SPLINE
SPL {X  -165.650, Y  +465.900, Z    +0.000, E1   -37.888, E3 +418401.268}
SPL {X  -165.650, Y  +471.256, Z    +0.000, E1   -37.789, E3 +418415.836}
SPL {X  -165.650, Y  +475.981, Z    +0.000, E1   -37.909, E3 +418427.559}
SPL {X  -165.650, Y  +481.142, Z    +0.000, E1   -37.875, E3 +418441.379}
SPL {X  -165.650, Y  +485.415, Z    +0.000, E1   -37.930, E3 +418452.144}
SPL {X  -165.650, Y  +488.381, Z    +0.000, E1   -37.932, E3 +418459.911}
SPL {X  -165.650, Y  +492.473, Z    +0.000, E1   -37.882, E3 +418471.081}
SPL {X  -165.650, Y  +496.967, Z    +0.000, E1   -37.731, E3 +418483.788}
SPL {X  -165.650, Y  +502.007, Z    +0.000, E1   -37.899, E3 +418496.077}
SPL {X  -165.650, Y  +506.838, Z    +0.000, E1   -38.018, E3 +418507.973}
SPL {X  -165.650, Y  +510.962, Z    +0.000, E1   -37.876, E3 +418519.687}
SPL {X  -165.650, Y  +513.924, Z    +0.000, E1   -37.557, E3 +418529.355}
SPL {X  -165.650, Y  +519.541, Z    +0.000, E1   -37.994, E3 +418541.689}
SPL {X  -165.650, Y  +524.168, Z    +0.000, E1   -37.816, E3 +418554.745}
SPL {X  -165.650, Y  +528.532, Z    +0.000, E1   -37.895, E3 +418565.811}
SPL {X  -165.650, Y  +532.864, Z    +0.000, E1   -37.846, E3 +418577.452}
SPL {X  -165.650, Y  +537.279, Z    +0.000, E1   -37.980, E3 +418588.275}
SPL {X  -165.650, Y  +540.651, Z    +0.000, E1   -37.651, E3 +418599.077}
SPL {X  -165.650, Y  +545.726, Z    +0.000, E1   -37.963, E3 +418610.643}
SPL {X  -165.650, Y  +550.427, Z    +0.000, E1   -37.784, E3 +418624.061}
SPL {X  -165.650, Y  +554.659, Z    +0.000, E1   -37.927, E3 +418634.245}
SPL {X  -165.650, Y  +557.856, Z    +0.000, E1   -37.998, E3 +418642.195}
SPL {X  -165.650, Y  +562.748, Z    +0.000, E1   -37.890, E3 +418655.937}
SPL {X  -165.650, Y  +567.848, Z    +0.000, E1   -37.954, E3 +418668.710}
SPL {X  -165.650, Y  +571.305, Z    +0.000, E1   -37.718, E3 +418679.371}
SPL {X  -165.650, Y  +577.754, Z    +0.000, E1   -38.006, E3 +418694.662}
SPL {X  -165.650, Y  +583.042, Z    +0.000, E1   -37.879, E3 +418709.206}
SPL {X  -165.650, Y  +587.643, Z    +0.000, E1   -37.879, E3 +418721.284}
SPL {X  -165.650, Y  +592.833, Z    +0.000, E1   -37.896, E3 +418734.932}
SPL {X  -165.650, Y  +597.119, Z    +0.000, E1   -37.642, E3 +418747.661}
SPL {X  -165.650, Y  +602.808, Z    +0.000, E1   -37.983, E3 +418760.668}
SPL {X  -165.650, Y  +607.937, Z    +0.000, E1   -37.862, E3 +418774.829}
SPL {X  -165.650, Y  +614.056, Z    +0.000, E1   -37.933, E3 +418790.600}
SPL {X  -165.650, Y  +619.142, Z    +0.000, E1   -37.954, E3 +418803.618}
SPL {X  -165.650, Y  +622.884, Z    +0.000, E1   -37.770, E3 +418814.661}
SPL {X  -165.650, Y  +628.759, Z    +0.000, E1   -37.993, E3 +418828.831}
SPL {X  -165.650, Y  +633.686, Z    +0.000, E1   -37.760, E3 +418843.106}
SPL {X  -165.650, Y  +639.918, Z    +0.000, E1   -37.892, E3 +418858.915}
SPL {X  -165.650, Y  +645.851, Z    +0.000, E1   -37.854, E3 +418874.567}
SPL {X  -165.650, Y  +650.450, Z    +0.000, E1   -37.924, E3 +418886.207}
SPL {X  -165.650, Y  +654.711, Z    +0.000, E1   -37.888, E3 +418897.641}
SPL {X  -165.650, Y  +660.285, Z    +0.000, E1   -37.928, E3 +418912.159}
SPL {X  -165.650, Y  +665.663, Z    +0.000, E1   -37.913, E3 +418926.247}
SPL {X  -165.650, Y  +669.913, Z    +0.000, E1   -37.905, E3 +418937.449}
SPL {X  -165.650, Y  +674.729, Z    +0.000, E1   -37.860, E3 +418950.458}
SPL {X  -165.591, Y  +679.928, Z    +0.000, E1   -37.818, E3 +418964.375}
SPL {X  -165.340, Y  +685.624, Z    +0.000, E1   -37.900, E3 +418978.910}
SPL {X  -165.010, Y  +690.051, Z    +0.000, E1   -37.675, E3 +418991.841}
SPL {X  -164.652, Y  +693.652, Z    +0.000, E1   -37.750, E3 +419000.771}
SPL {X  -164.143, Y  +697.797, Z    +0.000, E1   -37.636, E3 +419012.591}
SPL {X  -163.447, Y  +702.423, Z    +0.000, E1   -37.496, E3 +419025.399}
SPL {X  -162.809, Y  +706.049, Z    +0.000, E1   -37.384, E3 +419035.669}
SPL {X  -161.803, Y  +710.992, Z    +0.000, E1   -37.315, E3 +419049.134}
SPL {X  -160.993, Y  +714.501, Z    +0.000, E1   -36.839, E3 +419061.011}
SPL {X  -159.156, Y  +721.427, Z    +0.000, E1   -38.526, E3 +419069.089}
SPL {X  -144.831, Y  +755.898, Z    +0.000, E1   -42.981, E3 +419130.505}
ENDSPLINE

SPLINE
SPL {X  -153.047, Y  +738.876, Z    +0.000, E1   -33.363, E3 +419212.720}
SPL {X  -162.649, Y  +706.888, Z    +0.000, E1   -19.911, E3 +419202.081}
SPL {X  -165.011, Y  +690.033, Z    +0.000, E1   -11.292, E3 +419198.316}
SPL {X  -165.581, Y  +680.273, Z    +0.000, E1    -5.775, E3 +419194.114}
SPL {X  -165.650, Y  +674.660, Z    +0.000, E1    -2.196, E3 +419194.781}
SPL {X  -165.650, Y  +669.932, Z    +0.000, E1    +1.173, E3 +419193.357}
SPL {X  -165.650, Y  +665.412, Z    +0.000, E1    +4.953, E3 +419192.537}
SPL {X  -165.650, Y  +660.335, Z    +0.000, E1    +9.682, E3 +419193.054}
SPL {X  -165.650, Y  +650.970, Z    +0.000, E1   +18.783, E3 +419193.602}
SPL {X  -165.650, Y  +637.823, Z    +0.000, E1   +39.473, E3 +419173.703}
SPL {X  -165.650, Y  +613.283, Z    +0.000, E1   +49.826, E3 +419189.271}
SPL {X  -165.650, Y  +609.693, Z    +0.000, E1   +42.113, E3 +419217.405}
SPL {X  -165.650, Y  +571.120, Z    +0.000, E1   +47.704, E3 +419262.214}
ENDSPLINE

SPLINE
SPL {X  -165.650, Y  +586.477, Z    +0.000, E1   +39.172, E3 +419278.758}
ENDSPLINE

SPLINE
SPL {X  -165.650, Y  +581.917, Z    +0.000, E1   +39.019, E3 +419291.160}
SPL {X  -165.650, Y  +577.218, Z    +0.000, E1   +38.911, E3 +419303.701}
SPL {X  -165.650, Y  +572.890, Z    +0.000, E1   +39.033, E3 +419313.838}
SPL {X  -165.650, Y  +569.005, Z    +0.000, E1   +38.999, E3 +419323.929}
SPL {X  -165.650, Y  +564.604, Z    +0.000, E1   +38.986, E3 +419335.065}
SPL {X  -165.650, Y  +560.333, Z    +0.000, E1   +38.995, E3 +419345.830}
SPL {X  -165.650, Y  +556.690, Z    +0.000, E1   +39.061, E3 +419354.549}
SPL {X  -165.650, Y  +552.186, Z    +0.000, E1   +39.063, E3 +419366.067}
SPL {X  -165.650, Y  +547.091, Z    +0.000, E1   +39.070, E3 +419378.727}
SPL {X  -165.650, Y  +526.098, Z    +0.000, E1   +45.792, E3 +419385.794}
SPL {X  -165.650, Y  +510.223, Z    +0.000, E1   +49.521, E3 +419393.191}
SPL {X  -165.650, Y  +505.315, Z    +0.000, E1   +48.718, E3 +419407.000}
SPL {X  -165.650, Y  +499.987, Z    +0.000, E1   +47.980, E3 +419420.786}
SPL {X  -165.650, Y  +497.138, Z    +0.000, E1   +47.280, E3 +419430.279}
SPL {X  -165.650, Y  +493.273, Z    +0.000, E1   +46.518, E3 +419442.260}
SPL {X  -165.650, Y  +489.140, Z    +0.000, E1   +45.675, E3 +419455.387}
SPL {X  -165.650, Y  +485.420, Z    +0.000, E1   +44.711, E3 +419468.606}
SPL {X  -165.650, Y  +480.756, Z    +0.000, E1   +43.779, E3 +419484.084}
SPL {X  -165.650, Y  +475.837, Z    +0.000, E1   +42.787, E3 +419500.545}
SPL {X  -165.650, Y  +472.413, Z    +0.000, E1   +41.852, E3 +419513.660}
SPL {X  -165.650, Y  +469.721, Z    +0.000, E1   +41.361, E3 +419522.686}
SPL {X  -165.650, Y  +467.130, Z    +0.000, E1   +40.624, E3 +419533.368}
SPL {X  -165.650, Y  +463.869, Z    +0.000, E1   +39.839, E3 +419545.836}
SPL {X  -165.650, Y  +462.171, Z    +0.000, E1   +38.860, E3 +419556.015}
SPL {X  -165.650, Y  +457.119, Z    +0.000, E1   +39.087, E3 +419567.393}
SPL {X  -165.650, Y  +452.884, Z    +0.000, E1   +39.185, E3 +419577.441}
SPL {X  -165.650, Y  +449.593, Z    +0.000, E1   +38.852, E3 +419587.736}
SPL {X  -165.650, Y  +445.147, Z    +0.000, E1   +39.088, E3 +419597.558}
SPL {X  -165.650, Y  +439.751, Z    +0.000, E1   +39.254, E3 +419610.175}
SPL {X  -165.650, Y  +435.510, Z    +0.000, E1   +39.051, E3 +419621.987}
SPL {X  -165.650, Y  +430.832, Z    +0.000, E1   +39.105, E3 +419633.443}
SPL {X  -165.650, Y  +426.072, Z    +0.000, E1   +39.194, E3 +419644.866}
SPL {X  -165.650, Y  +422.372, Z    +0.000, E1   +38.952, E3 +419655.602}
SPL {X  -165.650, Y  +417.591, Z    +0.000, E1   +39.157, E3 +419666.455}
SPL {X  -165.650, Y  +412.842, Z    +0.000, E1   +39.072, E3 +419678.954}
SPL {X  -165.650, Y  +407.612, Z    +0.000, E1   +39.068, E3 +419692.127}
SPL {X  -165.650, Y  +402.767, Z    +0.000, E1   +39.122, E3 +419703.982}
SPL {X  -165.650, Y  +398.352, Z    +0.000, E1   +39.113, E3 +419715.135}
SPL {X  -165.650, Y  +393.915, Z    +0.000, E1   +39.126, E3 +419726.212}
SPL {X  -165.650, Y  +389.523, Z    +0.000, E1   +39.115, E3 +419737.322}
SPL {X  -165.650, Y  +384.404, Z    +0.000, E1   +39.147, E3 +419750.058}
SPL {X  -165.650, Y  +380.058, Z    +0.000, E1   +39.073, E3 +419761.345}
SPL {X  -165.624, Y  +375.547, Z    +0.000, E1   +39.047, E3 +419772.944}
SPL {X  -165.438, Y  +370.129, Z    +0.000, E1   +39.090, E3 +419786.330}
SPL {X  -165.143, Y  +365.555, Z    +0.000, E1   +39.161, E3 +419797.302}
SPL {X  -164.909, Y  +362.853, Z    +0.000, E1   +38.709, E3 +419806.849}
SPL {X  -164.359, Y  +357.858, Z    +0.000, E1   +39.066, E3 +419817.312}
SPL {X  -163.818, Y  +353.935, Z    +0.000, E1   +38.811, E3 +419828.706}
SPL {X  -163.055, Y  +349.296, Z    +0.000, E1   +38.669, E3 +419841.211}
SPL {X  -162.021, Y  +344.016, Z    +0.000, E1   +38.517, E3 +419855.500}
SPL {X  -160.588, Y  +337.861, Z    +0.000, E1   +38.304, E3 +419872.214}
SPL {X  -151.400, Y  +311.284, Z    +0.000, E1   +46.597, E3 +419883.823}
SPL {X  -145.363, Y  +299.068, Z    +0.000, E1   +42.035, E3 +419948.986}
ENDSPLINE

SPLINE
SPL {X  -147.808, Y  +303.715, Z    +0.000, E1   +39.616, E3 +419961.399}
SPL {X  -154.092, Y  +317.709, Z    +0.000, E1   +32.342, E3 +420026.112}
SPL {X  -161.950, Y  +343.684, Z    +0.000, E1   +21.785, E3 +420002.951}
SPL {X  -164.623, Y  +360.087, Z    +0.000, E1   +13.426, E3 +420011.602}
SPL {X  -165.588, Y  +373.983, Z    +0.000, E1    +5.738, E3 +420004.379}
SPL {X  -165.650, Y  +380.761, Z    +0.000, E1    +1.351, E3 +420006.103}
SPL {X  -165.650, Y  +386.484, Z    +0.000, E1    -2.972, E3 +420004.110}
SPL {X  -165.650, Y  +392.905, Z    +0.000, E1    -8.557, E3 +420006.164}
SPL {X  -165.650, Y  +404.146, Z    +0.000, E1   -20.514, E3 +420000.894}
SPL {X  -165.650, Y  +412.709, Z    +0.000, E1   -30.621, E3 +419995.857}
SPL {X  -165.650, Y  +437.337, Z    +0.000, E1   -46.817, E3 +420002.204}
SPL {X  -165.650, Y  +445.979, Z    +0.000, E1   -45.194, E3 +420020.273}
SPL {X  -165.650, Y  +459.839, Z    +0.000, E1   -48.128, E3 +420032.014}
SPL {X  -165.650, Y  +484.108, Z    +0.000, E1   -48.531, E3 +420069.005}
ENDSPLINE

SPLINE
SPL {X  -165.650, Y  +464.452, Z    +0.000, E1   -38.833, E3 +420084.066}
ENDSPLINE

SPLINE
SPL {X  -165.650, Y  +467.011, Z    +0.000, E1   -37.866, E3 +420096.490}
SPL {X  -165.650, Y  +471.256, Z    +0.000, E1   -37.789, E3 +420108.143}
SPL {X  -165.650, Y  +475.981, Z    +0.000, E1   -37.909, E3 +420119.866}
SPL {X  -165.650, Y  +481.142, Z    +0.000, E1   -37.875, E3 +420133.687}
SPL {X  -165.650, Y  +487.016, Z    +0.000, E1   -37.964, E3 +420148.592}
SPL {X  -165.650, Y  +492.473, Z    +0.000, E1   -37.882, E3 +420163.388}
SPL {X  -165.650, Y  +496.967, Z    +0.000, E1   -37.731, E3 +420176.095}
SPL {X  -165.650, Y  +502.007, Z    +0.000, E1   -37.899, E3 +420188.384}
SPL {X  -165.650, Y  +507.602, Z    +0.000, E1   -37.863, E3 +420203.414}
SPL {X  -165.650, Y  +513.428, Z    +0.000, E1   -37.892, E3 +420218.480}
SPL {X  -165.650, Y  +518.534, Z    +0.000, E1   -37.976, E3 +420231.343}
SPL {X  -165.650, Y  +523.331, Z    +0.000, E1   -37.880, E3 +420244.565}
SPL {X  -165.650, Y  +528.532, Z    +0.000, E1   -37.895, E3 +420258.119}
SPL {X  -165.650, Y  +534.316, Z    +0.000, E1   -37.926, E3 +420273.233}
SPL {X  -165.650, Y  +539.968, Z    +0.000, E1   -37.796, E3 +420288.820}
SPL {X  -165.650, Y  +545.726, Z    +0.000, E1   -37.963, E3 +420302.951}
SPL {X  -165.650, Y  +550.427, Z    +0.000, E1   -37.784, E3 +420316.369}
SPL {X  -165.650, Y  +556.372, Z    +0.000, E1   -37.998, E3 +420330.765}
SPL {X  -165.650, Y  +561.478, Z    +0.000, E1   -37.846, E3 +420345.012}
SPL {X  -165.650, Y  +566.625, Z    +0.000, E1   -37.932, E3 +420358.041}
SPL {X  -165.650, Y  +571.305, Z    +0.000, E1   -37.718, E3 +420371.679}
SPL {X  -165.650, Y  +577.754, Z    +0.000, E1   -38.006, E3 +420386.970}
SPL {X  -165.650, Y  +583.042, Z    +0.000, E1   -37.879, E3 +420401.514}
SPL {X  -165.650, Y  +587.643, Z    +0.000, E1   -37.879, E3 +420413.592}
SPL {X  -165.650, Y  +592.833, Z    +0.000, E1   -37.896, E3 +420427.240}
SPL {X  -165.650, Y  +597.119, Z    +0.000, E1   -37.642, E3 +420439.969}
SPL {X  -165.650, Y  +602.808, Z    +0.000, E1   -37.983, E3 +420452.975}
SPL {X  -165.650, Y  +607.937, Z    +0.000, E1   -37.862, E3 +420467.137}
SPL {X  -165.650, Y  +612.863, Z    +0.000, E1   -37.857, E3 +420480.109}
SPL {X  -165.650, Y  +618.208, Z    +0.000, E1   -37.992, E3 +420493.352}
SPL {X  -165.650, Y  +622.884, Z    +0.000, E1   -37.770, E3 +420506.969}
SPL {X  -165.650, Y  +628.759, Z    +0.000, E1   -37.993, E3 +420521.139}
SPL {X  -165.650, Y  +633.686, Z    +0.000, E1   -37.760, E3 +420535.414}
SPL {X  -165.650, Y  +639.918, Z    +0.000, E1   -37.892, E3 +420551.222}
SPL {X  -165.650, Y  +645.851, Z    +0.000, E1   -37.854, E3 +420566.875}
SPL {X  -165.650, Y  +650.450, Z    +0.000, E1   -37.924, E3 +420578.515}
SPL {X  -165.650, Y  +654.711, Z    +0.000, E1   -37.888, E3 +420589.949}
SPL {X  -165.650, Y  +658.674, Z    +0.000, E1   -37.902, E3 +420600.217}
SPL {X  -165.650, Y  +661.754, Z    +0.000, E1   -37.878, E3 +420608.453}
SPL {X  -165.650, Y  +665.663, Z    +0.000, E1   -37.913, E3 +420618.554}
SPL {X  -165.650, Y  +669.913, Z    +0.000, E1   -37.905, E3 +420629.756}
SPL {X  -165.650, Y  +674.729, Z    +0.000, E1   -37.860, E3 +420642.766}
SPL {X  -165.591, Y  +679.928, Z    +0.000, E1   -37.818, E3 +420656.683}
SPL {X  -165.340, Y  +685.624, Z    +0.000, E1   -37.900, E3 +420671.218}
SPL {X  -165.010, Y  +690.051, Z    +0.000, E1   -37.675, E3 +420684.149}
SPL {X  -164.376, Y  +696.008, Z    +0.000, E1   -37.753, E3 +420699.513}
SPL {X  -163.617, Y  +701.375, Z    +0.000, E1   -37.486, E3 +420715.106}
SPL {X  -162.809, Y  +706.049, Z    +0.000, E1   -37.384, E3 +420727.977}
SPL {X  -161.803, Y  +710.992, Z    +0.000, E1   -37.315, E3 +420741.442}
SPL {X  -160.993, Y  +714.501, Z    +0.000, E1   -36.839, E3 +420753.318}
SPL {X  -159.156, Y  +721.427, Z    +0.000, E1   -38.526, E3 +420761.396}
SPL {X  -144.831, Y  +755.898, Z    +0.000, E1   -42.981, E3 +420822.812}
ENDSPLINE

SPLINE
SPL {X  -153.047, Y  +738.876, Z    +0.000, E1   -33.363, E3 +420905.027}
SPL {X  -162.649, Y  +706.888, Z    +0.000, E1   -19.911, E3 +420894.389}
SPL {X  -165.011, Y  +690.033, Z    +0.000, E1   -11.292, E3 +420890.623}
SPL {X  -165.581, Y  +680.273, Z    +0.000, E1    -5.775, E3 +420886.422}
SPL {X  -165.650, Y  +673.781, Z    +0.000, E1    -1.642, E3 +420885.665}
SPL {X  -165.650, Y  +669.471, Z    +0.000, E1    +1.546, E3 +420886.819}
SPL {X  -165.650, Y  +665.412, Z    +0.000, E1    +4.953, E3 +420884.844}
SPL {X  -165.650, Y  +658.891, Z    +0.000, E1   +11.031, E3 +420885.155}
SPL {X  -165.650, Y  +649.186, Z    +0.000, E1   +20.530, E3 +420886.415}
SPL {X  -165.650, Y  +637.823, Z    +0.000, E1   +39.473, E3 +420866.011}
SPL {X  -165.650, Y  +614.460, Z    +0.000, E1   +51.116, E3 +420876.880}
SPL {X  -165.650, Y  +609.746, Z    +0.000, E1   +42.762, E3 +420907.538}
SPL {X  -165.650, Y  +571.120, Z    +0.000, E1   +47.704, E3 +420954.522}
ENDSPLINE

SPLINE
SPL {X  -165.650, Y  +586.477, Z    +0.000, E1   +39.172, E3 +420971.066}
ENDSPLINE

SPLINE
SPL {X  -165.650, Y  +581.917, Z    +0.000, E1   +39.019, E3 +420983.468}
SPL {X  -165.650, Y  +577.218, Z    +0.000, E1   +38.911, E3 +420996.008}
SPL {X  -165.650, Y  +572.890, Z    +0.000, E1   +39.033, E3 +421006.146}
SPL {X  -165.650, Y  +569.005, Z    +0.000, E1   +38.999, E3 +421016.237}
SPL {X  -165.650, Y  +564.604, Z    +0.000, E1   +38.986, E3 +421027.372}
SPL {X  -165.650, Y  +560.333, Z    +0.000, E1   +38.995, E3 +421038.138}
SPL {X  -165.650, Y  +554.558, Z    +0.000, E1   +39.065, E3 +421052.427}
SPL {X  -165.650, Y  +548.147, Z    +0.000, E1   +39.104, E3 +421068.283}
SPL {X  -165.650, Y  +526.098, Z    +0.000, E1   +45.792, E3 +421078.102}
SPL {X  -165.650, Y  +510.223, Z    +0.000, E1   +49.521, E3 +421085.499}
SPL {X  -165.650, Y  +506.429, Z    +0.000, E1   +48.913, E3 +421095.912}
SPL {X  -165.650, Y  +501.394, Z    +0.000, E1   +48.110, E3 +421109.891}
SPL {X  -165.650, Y  +497.138, Z    +0.000, E1   +47.280, E3 +421122.587}
SPL {X  -165.650, Y  +493.273, Z    +0.000, E1   +46.518, E3 +421134.568}
SPL {X  -165.650, Y  +489.140, Z    +0.000, E1   +45.675, E3 +421147.695}
SPL {X  -165.650, Y  +485.420, Z    +0.000, E1   +44.711, E3 +421160.914}
SPL {X  -165.650, Y  +482.261, Z    +0.000, E1   +43.960, E3 +421171.866}
SPL {X  -165.650, Y  +478.467, Z    +0.000, E1   +43.371, E3 +421183.693}
SPL {X  -165.650, Y  +474.990, Z    +0.000, E1   +42.535, E3 +421196.045}
SPL {X  -165.650, Y  +472.413, Z    +0.000, E1   +41.852, E3 +421205.967}
SPL {X  -165.650, Y  +469.721, Z    +0.000, E1   +41.361, E3 +421214.994}
SPL {X  -165.650, Y  +467.130, Z    +0.000, E1   +40.624, E3 +421225.676}
SPL {X  -165.650, Y  +463.869, Z    +0.000, E1   +39.839, E3 +421238.144}
SPL {X  -165.650, Y  +462.171, Z    +0.000, E1   +38.860, E3 +421248.323}
SPL {X  -165.650, Y  +457.119, Z    +0.000, E1   +39.087, E3 +421259.701}
SPL {X  -165.650, Y  +452.884, Z    +0.000, E1   +39.185, E3 +421269.749}
SPL {X  -165.650, Y  +449.593, Z    +0.000, E1   +38.852, E3 +421280.044}
SPL {X  -165.650, Y  +445.147, Z    +0.000, E1   +39.088, E3 +421289.866}
SPL {X  -165.650, Y  +439.751, Z    +0.000, E1   +39.254, E3 +421302.483}
SPL {X  -165.650, Y  +435.510, Z    +0.000, E1   +39.051, E3 +421314.294}
SPL {X  -165.650, Y  +430.832, Z    +0.000, E1   +39.105, E3 +421325.751}
SPL {X  -165.650, Y  +426.072, Z    +0.000, E1   +39.194, E3 +421337.174}
SPL {X  -165.650, Y  +422.372, Z    +0.000, E1   +38.952, E3 +421347.910}
SPL {X  -165.650, Y  +416.355, Z    +0.000, E1   +39.151, E3 +421362.070}
SPL {X  -165.650, Y  +408.927, Z    +0.000, E1   +39.115, E3 +421381.029}
SPL {X  -165.650, Y  +402.767, Z    +0.000, E1   +39.122, E3 +421396.290}
SPL {X  -165.650, Y  +398.352, Z    +0.000, E1   +39.113, E3 +421407.443}
SPL {X  -165.650, Y  +393.915, Z    +0.000, E1   +39.126, E3 +421418.520}
SPL {X  -165.650, Y  +388.386, Z    +0.000, E1   +39.140, E3 +421432.470}
SPL {X  -165.650, Y  +383.342, Z    +0.000, E1   +39.144, E3 +421444.956}
SPL {X  -165.650, Y  +378.675, Z    +0.000, E1   +39.090, E3 +421457.174}
SPL {X  -165.597, Y  +374.311, Z    +0.000, E1   +39.013, E3 +421468.460}
SPL {X  -165.438, Y  +370.129, Z    +0.000, E1   +39.090, E3 +421478.638}
SPL {X  -165.143, Y  +365.555, Z    +0.000, E1   +39.161, E3 +421489.610}
SPL {X  -164.909, Y  +362.853, Z    +0.000, E1   +38.709, E3 +421499.156}
SPL {X  -164.359, Y  +357.858, Z    +0.000, E1   +39.066, E3 +421509.619}
SPL {X  -163.818, Y  +353.935, Z    +0.000, E1   +38.811, E3 +421521.014}
SPL {X  -163.055, Y  +349.296, Z    +0.000, E1   +38.669, E3 +421533.519}
SPL {X  -162.021, Y  +344.016, Z    +0.000, E1   +38.517, E3 +421547.808}
SPL {X  -160.588, Y  +337.861, Z    +0.000, E1   +38.304, E3 +421564.522}
SPL {X  -151.400, Y  +311.284, Z    +0.000, E1   +46.597, E3 +421576.131}
SPL {X  -145.363, Y  +299.068, Z    +0.000, E1   +42.035, E3 +421641.293}
ENDSPLINE

SPLINE
SPL {X  -147.808, Y  +303.715, Z    +0.000, E1   +39.616, E3 +421653.707}
SPL {X  -154.092, Y  +317.709, Z    +0.000, E1   +32.342, E3 +421718.420}
SPL {X  -161.950, Y  +343.684, Z    +0.000, E1   +21.785, E3 +421695.259}
SPL {X  -164.623, Y  +360.087, Z    +0.000, E1   +13.426, E3 +421703.909}
SPL {X  -165.588, Y  +373.983, Z    +0.000, E1    +5.738, E3 +421696.686}
SPL {X  -165.650, Y  +380.761, Z    +0.000, E1    +1.351, E3 +421698.410}
SPL {X  -165.650, Y  +386.484, Z    +0.000, E1    -2.972, E3 +421696.417}
SPL {X  -165.650, Y  +392.905, Z    +0.000, E1    -8.557, E3 +421698.471}
SPL {X  -165.650, Y  +404.146, Z    +0.000, E1   -20.514, E3 +421693.201}
SPL {X  -165.650, Y  +416.920, Z    +0.000, E1   -34.832, E3 +421687.164}
SPL {X  -165.650, Y  +445.455, Z    +0.000, E1   -46.044, E3 +421709.255}
SPL {X  -165.650, Y  +459.839, Z    +0.000, E1   -48.128, E3 +421724.321}
SPL {X  -165.650, Y  +484.108, Z    +0.000, E1   -48.531, E3 +421761.313}
ENDSPLINE

SPLINE
SPL {X  -165.650, Y  +464.452, Z    +0.000, E1   -38.833, E3 +421776.374}
ENDSPLINE

SPLINE
SPL {X  -165.650, Y  +467.011, Z    +0.000, E1   -37.866, E3 +421788.797}
SPL {X  -165.650, Y  +471.256, Z    +0.000, E1   -37.789, E3 +421800.451}
SPL {X  -165.650, Y  +475.981, Z    +0.000, E1   -37.909, E3 +421812.174}
SPL {X  -165.650, Y  +481.142, Z    +0.000, E1   -37.875, E3 +421825.994}
SPL {X  -165.650, Y  +487.016, Z    +0.000, E1   -37.964, E3 +421840.900}
SPL {X  -165.650, Y  +492.473, Z    +0.000, E1   -37.882, E3 +421855.696}
SPL {X  -165.650, Y  +496.967, Z    +0.000, E1   -37.731, E3 +421868.403}
SPL {X  -165.650, Y  +502.007, Z    +0.000, E1   -37.899, E3 +421880.692}
SPL {X  -165.650, Y  +506.838, Z    +0.000, E1   -38.018, E3 +421892.589}
SPL {X  -165.650, Y  +510.962, Z    +0.000, E1   -37.876, E3 +421904.303}
SPL {X  -165.650, Y  +516.973, Z    +0.000, E1   -37.871, E3 +421920.330}
SPL {X  -165.650, Y  +523.331, Z    +0.000, E1   -37.880, E3 +421936.873}
SPL {X  -165.650, Y  +528.532, Z    +0.000, E1   -37.895, E3 +421950.426}
SPL {X  -165.650, Y  +532.864, Z    +0.000, E1   -37.846, E3 +421962.068}
SPL {X  -165.650, Y  +537.279, Z    +0.000, E1   -37.980, E3 +421972.890}
SPL {X  -165.650, Y  +540.651, Z    +0.000, E1   -37.651, E3 +421983.693}
SPL {X  -165.650, Y  +545.726, Z    +0.000, E1   -37.963, E3 +421995.258}
SPL {X  -165.650, Y  +550.427, Z    +0.000, E1   -37.784, E3 +422008.676}
SPL {X  -165.650, Y  +556.372, Z    +0.000, E1   -37.998, E3 +422023.072}
SPL {X  -165.650, Y  +561.478, Z    +0.000, E1   -37.846, E3 +422037.320}
SPL {X  -165.650, Y  +566.625, Z    +0.000, E1   -37.932, E3 +422050.349}
SPL {X  -165.650, Y  +571.305, Z    +0.000, E1   -37.718, E3 +422063.986}
SPL {X  -165.650, Y  +576.676, Z    +0.000, E1   -38.057, E3 +422075.983}
SPL {X  -165.650, Y  +581.909, Z    +0.000, E1   -37.903, E3 +422090.854}
SPL {X  -165.650, Y  +587.643, Z    +0.000, E1   -37.879, E3 +422105.899}
SPL {X  -165.650, Y  +592.833, Z    +0.000, E1   -37.896, E3 +422119.548}
SPL {X  -165.650, Y  +597.119, Z    +0.000, E1   -37.642, E3 +422132.277}
SPL {X  -165.650, Y  +602.808, Z    +0.000, E1   -37.983, E3 +422145.283}
SPL {X  -165.650, Y  +607.937, Z    +0.000, E1   -37.862, E3 +422159.444}
SPL {X  -165.650, Y  +614.056, Z    +0.000, E1   -37.933, E3 +422175.215}
SPL {X  -165.650, Y  +619.142, Z    +0.000, E1   -37.954, E3 +422188.234}
SPL {X  -165.650, Y  +622.884, Z    +0.000, E1   -37.770, E3 +422199.277}
SPL {X  -165.650, Y  +628.759, Z    +0.000, E1   -37.993, E3 +422213.446}
SPL {X  -165.650, Y  +633.686, Z    +0.000, E1   -37.760, E3 +422227.722}
SPL {X  -165.650, Y  +638.669, Z    +0.000, E1   -37.941, E3 +422239.728}
SPL {X  -165.650, Y  +643.208, Z    +0.000, E1   -37.786, E3 +422252.645}
SPL {X  -165.650, Y  +649.293, Z    +0.000, E1   -37.920, E3 +422267.935}
SPL {X  -165.650, Y  +654.711, Z    +0.000, E1   -37.888, E3 +422282.257}
SPL {X  -165.650, Y  +660.285, Z    +0.000, E1   -37.928, E3 +422296.775}
SPL {X  -165.650, Y  +665.663, Z    +0.000, E1   -37.913, E3 +422310.862}
SPL {X  -165.650, Y  +669.913, Z    +0.000, E1   -37.905, E3 +422322.064}
SPL {X  -165.650, Y  +674.729, Z    +0.000, E1   -37.860, E3 +422335.074}
SPL {X  -165.554, Y  +681.132, Z    +0.000, E1   -37.883, E3 +422351.908}
SPL {X  -165.277, Y  +686.615, Z    +0.000, E1   -37.853, E3 +422366.290}
SPL {X  -164.889, Y  +691.361, Z    +0.000, E1   -37.742, E3 +422379.644}
SPL {X  -164.246, Y  +697.018, Z    +0.000, E1   -37.690, E3 +422394.686}
SPL {X  -163.617, Y  +701.375, Z    +0.000, E1   -37.486, E3 +422407.413}
SPL {X  -162.809, Y  +706.049, Z    +0.000, E1   -37.384, E3 +422420.285}
SPL {X  -161.803, Y  +710.992, Z    +0.000, E1   -37.315, E3 +422433.749}
SPL {X  -160.993, Y  +714.501, Z    +0.000, E1   -36.839, E3 +422445.626}
SPL {X  -159.156, Y  +721.427, Z    +0.000, E1   -38.526, E3 +422453.704}
SPL {X  -144.831, Y  +755.898, Z    +0.000, E1   -42.981, E3 +422515.120}
ENDSPLINE

SPLINE
SPL {X  -153.047, Y  +738.876, Z    +0.000, E1   -33.363, E3 +422597.335}
SPL {X  -162.649, Y  +706.888, Z    +0.000, E1   -19.911, E3 +422586.697}
SPL {X  -165.011, Y  +690.033, Z    +0.000, E1   -11.292, E3 +422582.931}
SPL {X  -165.581, Y  +680.273, Z    +0.000, E1    -5.775, E3 +422578.729}
SPL {X  -165.650, Y  +674.660, Z    +0.000, E1    -2.196, E3 +422579.396}
SPL {X  -165.650, Y  +669.932, Z    +0.000, E1    +1.173, E3 +422577.973}
SPL {X  -165.650, Y  +665.412, Z    +0.000, E1    +4.953, E3 +422577.152}
SPL {X  -165.650, Y  +658.891, Z    +0.000, E1   +11.031, E3 +422577.463}
SPL {X  -165.650, Y  +649.186, Z    +0.000, E1   +20.530, E3 +422578.723}
SPL {X  -165.650, Y  +637.823, Z    +0.000, E1   +39.473, E3 +422558.319}
SPL {X  -165.650, Y  +614.460, Z    +0.000, E1   +51.116, E3 +422569.187}
SPL {X  -165.650, Y  +609.746, Z    +0.000, E1   +42.762, E3 +422599.845}
SPL {X  -165.650, Y  +571.120, Z    +0.000, E1   +47.704, E3 +422646.829}
ENDSPLINE

SPLINE
SPL {X  -165.650, Y  +586.477, Z    +0.000, E1   +39.172, E3 +422663.374}
ENDSPLINE

SPLINE
SPL {X  -165.650, Y  +581.917, Z    +0.000, E1   +39.019, E3 +422675.776}
SPL {X  -165.650, Y  +577.218, Z    +0.000, E1   +38.911, E3 +422688.316}
SPL {X  -165.650, Y  +572.890, Z    +0.000, E1   +39.033, E3 +422698.454}
SPL {X  -165.650, Y  +569.005, Z    +0.000, E1   +38.999, E3 +422708.544}
SPL {X  -165.650, Y  +564.604, Z    +0.000, E1   +38.986, E3 +422719.680}
SPL {X  -165.650, Y  +558.931, Z    +0.000, E1   +39.059, E3 +422733.748}
SPL {X  -165.650, Y  +553.380, Z    +0.000, E1   +39.004, E3 +422747.911}
SPL {X  -165.650, Y  +548.147, Z    +0.000, E1   +39.104, E3 +422760.591}
SPL {X  -165.650, Y  +526.098, Z    +0.000, E1   +45.792, E3 +422770.409}
SPL {X  -165.650, Y  +510.223, Z    +0.000, E1   +49.521, E3 +422777.807}
SPL {X  -165.650, Y  +506.429, Z    +0.000, E1   +48.913, E3 +422788.219}
SPL {X  -165.650, Y  +501.394, Z    +0.000, E1   +48.110, E3 +422802.198}
SPL {X  -165.650, Y  +497.138, Z    +0.000, E1   +47.280, E3 +422814.895}
SPL {X  -165.650, Y  +493.273, Z    +0.000, E1   +46.518, E3 +422826.875}
SPL {X  -165.650, Y  +489.140, Z    +0.000, E1   +45.675, E3 +422840.003}
SPL {X  -165.650, Y  +485.420, Z    +0.000, E1   +44.711, E3 +422853.222}
SPL {X  -165.650, Y  +480.756, Z    +0.000, E1   +43.779, E3 +422868.700}
SPL {X  -165.650, Y  +475.837, Z    +0.000, E1   +42.787, E3 +422885.160}
SPL {X  -165.650, Y  +472.413, Z    +0.000, E1   +41.852, E3 +422898.275}
SPL {X  -165.650, Y  +468.649, Z    +0.000, E1   +41.090, E3 +422911.639}
SPL {X  -165.650, Y  +464.675, Z    +0.000, E1   +40.045, E3 +422927.416}
SPL {X  -165.650, Y  +462.171, Z    +0.000, E1   +38.860, E3 +422940.631}
SPL {X  -165.650, Y  +457.119, Z    +0.000, E1   +39.087, E3 +422952.009}
SPL {X  -165.650, Y  +452.884, Z    +0.000, E1   +39.185, E3 +422962.057}
SPL {X  -165.650, Y  +449.593, Z    +0.000, E1   +38.852, E3 +422972.351}
SPL {X  -165.650, Y  +445.147, Z    +0.000, E1   +39.088, E3 +422982.174}
SPL {X  -165.650, Y  +439.751, Z    +0.000, E1   +39.254, E3 +422994.791}
SPL {X  -165.650, Y  +435.510, Z    +0.000, E1   +39.051, E3 +423006.602}
SPL {X  -165.650, Y  +430.832, Z    +0.000, E1   +39.105, E3 +423018.059}
SPL {X  -165.650, Y  +426.072, Z    +0.000, E1   +39.194, E3 +423029.482}
SPL {X  -165.650, Y  +422.372, Z    +0.000, E1   +38.952, E3 +423040.218}
SPL {X  -165.650, Y  +417.591, Z    +0.000, E1   +39.157, E3 +423051.071}
SPL {X  -165.650, Y  +412.842, Z    +0.000, E1   +39.072, E3 +423063.569}
SPL {X  -165.650, Y  +407.612, Z    +0.000, E1   +39.068, E3 +423076.742}
SPL {X  -165.650, Y  +402.767, Z    +0.000, E1   +39.122, E3 +423088.598}
SPL {X  -165.650, Y  +398.352, Z    +0.000, E1   +39.113, E3 +423099.750}
SPL {X  -165.650, Y  +393.915, Z    +0.000, E1   +39.126, E3 +423110.828}
SPL {X  -165.650, Y  +388.386, Z    +0.000, E1   +39.140, E3 +423124.777}
SPL {X  -165.650, Y  +383.342, Z    +0.000, E1   +39.144, E3 +423137.264}
SPL {X  -165.650, Y  +378.675, Z    +0.000, E1   +39.090, E3 +423149.482}
SPL {X  -165.597, Y  +374.311, Z    +0.000, E1   +39.013, E3 +423160.768}
SPL {X  -165.438, Y  +370.129, Z    +0.000, E1   +39.090, E3 +423170.945}
SPL {X  -165.143, Y  +365.555, Z    +0.000, E1   +39.161, E3 +423181.918}
SPL {X  -164.909, Y  +362.853, Z    +0.000, E1   +38.709, E3 +423191.464}
SPL {X  -164.359, Y  +357.858, Z    +0.000, E1   +39.066, E3 +423201.927}
SPL {X  -163.818, Y  +353.935, Z    +0.000, E1   +38.811, E3 +423213.321}
SPL {X  -163.055, Y  +349.296, Z    +0.000, E1   +38.669, E3 +423225.826}
SPL {X  -162.319, Y  +345.445, Z    +0.000, E1   +38.490, E3 +423236.522}
SPL {X  -161.279, Y  +340.696, Z    +0.000, E1   +38.442, E3 +423248.849}
SPL {X  -160.251, Y  +336.552, Z    +0.000, E1   +38.166, E3 +423260.715}
SPL {X  -151.400, Y  +311.284, Z    +0.000, E1   +46.597, E3 +423268.439}
SPL {X  -146.894, Y  +301.936, Z    +0.000, E1   +40.559, E3 +423341.603}
ENDSPLINE

SPLINE
SPL {X  -154.092, Y  +317.709, Z    +0.000, E1   +32.342, E3 +423410.727}
SPL {X  -161.950, Y  +343.684, Z    +0.000, E1   +21.785, E3 +423387.567}
SPL {X  -164.623, Y  +360.087, Z    +0.000, E1   +13.426, E3 +423396.217}
SPL {X  -165.489, Y  +371.187, Z    +0.000, E1    +7.370, E3 +423387.058}
SPL {X  -165.621, Y  +375.403, Z    +0.000, E1    +4.810, E3 +423389.956}
SPL {X  -165.650, Y  +380.761, Z    +0.000, E1    +1.351, E3 +423390.718}
SPL {X  -165.650, Y  +386.484, Z    +0.000, E1    -2.972, E3 +423388.725}
SPL {X  -165.650, Y  +392.905, Z    +0.000, E1    -8.557, E3 +423390.779}
SPL {X  -165.650, Y  +404.146, Z    +0.000, E1   -20.514, E3 +423385.509}
SPL {X  -165.650, Y  +412.709, Z    +0.000, E1   -30.621, E3 +423380.473}
SPL {X  -165.650, Y  +437.337, Z    +0.000, E1   -46.817, E3 +423386.820}
SPL {X  -165.650, Y  +450.640, Z    +0.000, E1   -46.274, E3 +423408.842}
SPL {X  -165.650, Y  +484.108, Z    +0.000, E1   -48.531, E3 +423453.621}
ENDSPLINE

SPLINE
SPL {X  -165.650, Y  +464.452, Z    +0.000, E1   -38.833, E3 +423468.681}
ENDSPLINE

SPLINE
SPL {X  -165.650, Y  +467.011, Z    +0.000, E1   -37.866, E3 +423481.105}
SPL {X  -165.650, Y  +471.256, Z    +0.000, E1   -37.789, E3 +423492.759}
SPL {X  -165.650, Y  +475.981, Z    +0.000, E1   -37.909, E3 +423504.482}
SPL {X  -165.650, Y  +481.142, Z    +0.000, E1   -37.875, E3 +423518.302}
SPL {X  -165.650, Y  +487.016, Z    +0.000, E1   -37.964, E3 +423533.207}
SPL {X  -165.650, Y  +492.473, Z    +0.000, E1   -37.882, E3 +423548.004}
SPL {X  -165.650, Y  +496.967, Z    +0.000, E1   -37.731, E3 +423560.711}
SPL {X  -165.650, Y  +502.007, Z    +0.000, E1   -37.899, E3 +423573.000}
SPL {X  -165.650, Y  +507.602, Z    +0.000, E1   -37.863, E3 +423588.030}
SPL {X  -165.650, Y  +513.428, Z    +0.000, E1   -37.892, E3 +423603.096}
SPL {X  -165.650, Y  +518.534, Z    +0.000, E1   -37.976, E3 +423615.959}
SPL {X  -165.650, Y  +523.331, Z    +0.000, E1   -37.880, E3 +423629.180}
SPL {X  -165.650, Y  +528.532, Z    +0.000, E1   -37.895, E3 +423642.734}
SPL {X  -165.650, Y  +532.864, Z    +0.000, E1   -37.846, E3 +423654.375}
SPL {X  -165.650, Y  +537.279, Z    +0.000, E1   -37.980, E3 +423665.198}
SPL {X  -165.650, Y  +540.651, Z    +0.000, E1   -37.651, E3 +423676.000}
SPL {X  -165.650, Y  +545.726, Z    +0.000, E1   -37.963, E3 +423687.566}
SPL {X  -165.650, Y  +550.427, Z    +0.000, E1   -37.784, E3 +423700.984}
SPL {X  -165.650, Y  +554.659, Z    +0.000, E1   -37.927, E3 +423711.168}
SPL {X  -165.650, Y  +557.856, Z    +0.000, E1   -37.998, E3 +423719.118}
SPL {X  -165.650, Y  +562.748, Z    +0.000, E1   -37.890, E3 +423732.861}
SPL {X  -165.650, Y  +567.848, Z    +0.000, E1   -37.954, E3 +423745.633}
SPL {X  -165.650, Y  +571.305, Z    +0.000, E1   -37.718, E3 +423756.294}
SPL {X  -165.650, Y  +577.754, Z    +0.000, E1   -38.006, E3 +423771.585}
SPL {X  -165.650, Y  +583.042, Z    +0.000, E1   -37.879, E3 +423786.129}
SPL {X  -165.650, Y  +587.643, Z    +0.000, E1   -37.879, E3 +423798.207}
SPL {X  -165.650, Y  +592.833, Z    +0.000, E1   -37.896, E3 +423811.856}
SPL {X  -165.650, Y  +599.187, Z    +0.000, E1   -37.841, E3 +423828.994}
SPL {X  -165.650, Y  +604.276, Z    +0.000, E1   -37.917, E3 +423841.681}
SPL {X  -165.650, Y  +607.937, Z    +0.000, E1   -37.862, E3 +423851.752}
SPL {X  -165.650, Y  +612.863, Z    +0.000, E1   -37.857, E3 +423864.725}
SPL {X  -165.650, Y  +618.208, Z    +0.000, E1   -37.992, E3 +423877.967}
SPL {X  -165.650, Y  +622.884, Z    +0.000, E1   -37.770, E3 +423891.584}
SPL {X  -165.650, Y  +628.759, Z    +0.000, E1   -37.993, E3 +423905.754}
SPL {X  -165.650, Y  +633.686, Z    +0.000, E1   -37.760, E3 +423920.029}
SPL {X  -165.650, Y  +638.669, Z    +0.000, E1   -37.941, E3 +423932.036}
SPL {X  -165.650, Y  +644.441, Z    +0.000, E1   -37.838, E3 +423948.051}
SPL {X  -165.650, Y  +650.450, Z    +0.000, E1   -37.924, E3 +423963.130}
SPL {X  -165.650, Y  +654.711, Z    +0.000, E1   -37.888, E3 +423974.564}
SPL {X  -165.650, Y  +660.285, Z    +0.000, E1   -37.928, E3 +423989.082}
SPL {X  -165.650, Y  +665.663, Z    +0.000, E1   -37.913, E3 +424003.170}
SPL {X  -165.650, Y  +671.321, Z    +0.000, E1   -37.904, E3 +424018.271}
SPL {X  -165.649, Y  +676.172, Z    +0.000, E1   -37.873, E3 +424030.968}
SPL {X  -165.554, Y  +681.132, Z    +0.000, E1   -37.883, E3 +424044.216}
SPL {X  -165.277, Y  +686.615, Z    +0.000, E1   -37.853, E3 +424058.598}
SPL {X  -165.010, Y  +690.051, Z    +0.000, E1   -37.675, E3 +424068.764}
SPL {X  -164.652, Y  +693.652, Z    +0.000, E1   -37.750, E3 +424077.694}
SPL {X  -164.143, Y  +697.797, Z    +0.000, E1   -37.636, E3 +424089.514}
SPL {X  -163.447, Y  +702.423, Z    +0.000, E1   -37.496, E3 +424102.322}
SPL {X  -162.809, Y  +706.049, Z    +0.000, E1   -37.384, E3 +424112.592}
SPL {X  -162.124, Y  +709.497, Z    +0.000, E1   -37.325, E3 +424121.915}
SPL {X  -161.242, Y  +713.462, Z    +0.000, E1   -37.074, E3 +424134.036}
SPL {X  -159.156, Y  +721.427, Z    +0.000, E1   -38.526, E3 +424146.012}
SPL {X  -144.831, Y  +755.898, Z    +0.000, E1   -42.981, E3 +424207.428}
ENDSPLINE

SPLINE
SPL {X  -153.047, Y  +738.876, Z    +0.000, E1   -33.363, E3 +424289.643}
SPL {X  -162.649, Y  +706.888, Z    +0.000, E1   -19.911, E3 +424279.004}
SPL {X  -165.011, Y  +690.033, Z    +0.000, E1   -11.292, E3 +424275.239}
SPL {X  -165.581, Y  +680.273, Z    +0.000, E1    -5.775, E3 +424271.037}
SPL {X  -165.650, Y  +674.660, Z    +0.000, E1    -2.196, E3 +424271.704}
SPL {X  -165.650, Y  +669.932, Z    +0.000, E1    +1.173, E3 +424270.280}
SPL {X  -165.650, Y  +665.412, Z    +0.000, E1    +4.953, E3 +424269.460}
SPL {X  -165.650, Y  +658.891, Z    +0.000, E1   +11.031, E3 +424269.770}
SPL {X  -165.650, Y  +649.186, Z    +0.000, E1   +20.530, E3 +424271.031}
SPL {X  -165.650, Y  +637.823, Z    +0.000, E1   +39.473, E3 +424250.627}
SPL {X  -165.650, Y  +614.460, Z    +0.000, E1   +51.116, E3 +424261.495}
SPL {X  -165.650, Y  +609.746, Z    +0.000, E1   +42.762, E3 +424292.153}
SPL {X  -165.650, Y  +571.120, Z    +0.000, E1   +47.704, E3 +424339.137}
ENDSPLINE

SPLINE
SPL {X  -165.650, Y  +586.477, Z    +0.000, E1   +39.172, E3 +424355.681}
ENDSPLINE

SPLINE
SPL {X  -165.650, Y  +581.917, Z    +0.000, E1   +39.019, E3 +424368.083}
SPL {X  -165.650, Y  +577.218, Z    +0.000, E1   +38.911, E3 +424380.624}
SPL {X  -165.650, Y  +571.720, Z    +0.000, E1   +39.004, E3 +424394.016}
SPL {X  -165.650, Y  +565.656, Z    +0.000, E1   +39.042, E3 +424409.125}
SPL {X  -165.650, Y  +560.333, Z    +0.000, E1   +38.995, E3 +424422.753}
SPL {X  -165.650, Y  +554.558, Z    +0.000, E1   +39.065, E3 +424437.042}
SPL {X  -165.650, Y  +548.147, Z    +0.000, E1   +39.104, E3 +424452.898}
SPL {X  -165.650, Y  +526.098, Z    +0.000, E1   +45.792, E3 +424462.717}
SPL {X  -165.650, Y  +510.223, Z    +0.000, E1   +49.521, E3 +424470.114}
SPL {X  -165.650, Y  +506.429, Z    +0.000, E1   +48.913, E3 +424480.527}
SPL {X  -165.650, Y  +501.394, Z    +0.000, E1   +48.110, E3 +424494.506}
SPL {X  -165.650, Y  +497.138, Z    +0.000, E1   +47.280, E3 +424507.202}
SPL {X  -165.650, Y  +493.273, Z    +0.000, E1   +46.518, E3 +424519.183}
SPL {X  -165.650, Y  +490.148, Z    +0.000, E1   +45.850, E3 +424529.127}
SPL {X  -165.650, Y  +486.159, Z    +0.000, E1   +44.975, E3 +424542.673}
SPL {X  -165.650, Y  +482.261, Z    +0.000, E1   +43.960, E3 +424556.481}
SPL {X  -165.650, Y  +479.614, Z    +0.000, E1   +43.544, E3 +424564.616}
SPL {X  -165.650, Y  +475.837, Z    +0.000, E1   +42.787, E3 +424577.468}
SPL {X  -165.650, Y  +472.413, Z    +0.000, E1   +41.852, E3 +424590.583}
SPL {X  -165.650, Y  +468.649, Z    +0.000, E1   +41.090, E3 +424603.946}
SPL {X  -165.650, Y  +464.675, Z    +0.000, E1   +40.045, E3 +424619.724}
SPL {X  -165.650, Y  +462.171, Z    +0.000, E1   +38.860, E3 +424632.938}
SPL {X  -165.650, Y  +457.119, Z    +0.000, E1   +39.087, E3 +424644.316}
SPL {X  -165.650, Y  +452.884, Z    +0.000, E1   +39.185, E3 +424654.364}
SPL {X  -165.650, Y  +449.593, Z    +0.000, E1   +38.852, E3 +424664.659}
SPL {X  -165.650, Y  +443.672, Z    +0.000, E1   +39.218, E3 +424677.508}
SPL {X  -165.650, Y  +436.874, Z    +0.000, E1   +39.135, E3 +424695.179}
SPL {X  -165.650, Y  +430.832, Z    +0.000, E1   +39.105, E3 +424710.366}
SPL {X  -165.650, Y  +426.072, Z    +0.000, E1   +39.194, E3 +424721.789}
SPL {X  -165.650, Y  +422.372, Z    +0.000, E1   +38.952, E3 +424732.525}
SPL {X  -165.650, Y  +417.591, Z    +0.000, E1   +39.157, E3 +424743.378}
SPL {X  -165.650, Y  +412.842, Z    +0.000, E1   +39.072, E3 +424755.877}
SPL {X  -165.650, Y  +407.612, Z    +0.000, E1   +39.068, E3 +424769.050}
SPL {X  -165.650, Y  +402.767, Z    +0.000, E1   +39.122, E3 +424780.905}
SPL {X  -165.650, Y  +398.352, Z    +0.000, E1   +39.113, E3 +424792.058}
SPL {X  -165.650, Y  +393.915, Z    +0.000, E1   +39.126, E3 +424803.135}
SPL {X  -165.650, Y  +389.523, Z    +0.000, E1   +39.115, E3 +424814.245}
SPL {X  -165.650, Y  +384.404, Z    +0.000, E1   +39.147, E3 +424826.981}
SPL {X  -165.650, Y  +380.058, Z    +0.000, E1   +39.073, E3 +424838.268}
SPL {X  -165.624, Y  +375.547, Z    +0.000, E1   +39.047, E3 +424849.867}
SPL {X  -165.438, Y  +370.129, Z    +0.000, E1   +39.090, E3 +424863.253}
SPL {X  -165.143, Y  +365.555, Z    +0.000, E1   +39.161, E3 +424874.225}
SPL {X  -164.909, Y  +362.853, Z    +0.000, E1   +38.709, E3 +424883.772}
SPL {X  -164.359, Y  +357.858, Z    +0.000, E1   +39.066, E3 +424894.235}
SPL {X  -163.818, Y  +353.935, Z    +0.000, E1   +38.811, E3 +424905.629}
SPL {X  -163.055, Y  +349.296, Z    +0.000, E1   +38.669, E3 +424918.134}
SPL {X  -162.021, Y  +344.016, Z    +0.000, E1   +38.517, E3 +424932.424}
SPL {X  -160.588, Y  +337.861, Z    +0.000, E1   +38.304, E3 +424949.137}
SPL {X  -153.716, Y  +316.763, Z    +0.000, E1   +45.637, E3 +424955.641}
SPL {X  -149.011, Y  +306.142, Z    +0.000, E1   +47.422, E3 +424965.673}
SPL {X  -146.894, Y  +301.936, Z    +0.000, E1   +40.559, E3 +425033.911}
ENDSPLINE

SPLINE
SPL {X  -154.092, Y  +317.709, Z    +0.000, E1   +32.342, E3 +425103.035}
SPL {X  -161.950, Y  +343.684, Z    +0.000, E1   +21.785, E3 +425079.874}
SPL {X  -164.623, Y  +360.087, Z    +0.000, E1   +13.426, E3 +425088.525}
SPL {X  -165.588, Y  +373.983, Z    +0.000, E1    +5.738, E3 +425081.302}
SPL {X  -165.650, Y  +380.761, Z    +0.000, E1    +1.351, E3 +425083.026}
SPL {X  -165.650, Y  +386.484, Z    +0.000, E1    -2.972, E3 +425081.033}
SPL {X  -165.650, Y  +391.786, Z    +0.000, E1    -7.566, E3 +425083.428}
SPL {X  -165.650, Y  +399.284, Z    +0.000, E1   -15.403, E3 +425078.613}
SPL {X  -165.650, Y  +409.824, Z    +0.000, E1   -26.455, E3 +425076.492}
SPL {X  -165.650, Y  +437.337, Z    +0.000, E1   -46.817, E3 +425079.128}
SPL {X  -165.650, Y  +445.979, Z    +0.000, E1   -45.194, E3 +425097.196}
SPL {X  -165.650, Y  +459.839, Z    +0.000, E1   -48.128, E3 +425108.937}
SPL {X  -165.650, Y  +484.108, Z    +0.000, E1   -48.531, E3 +425145.928}
ENDSPLINE

SPLINE
SPL {X  -165.650, Y  +464.452, Z    +0.000, E1   -38.833, E3 +425160.989}
ENDSPLINE

SPLINE
SPL {X  -165.650, Y  +467.011, Z    +0.000, E1   -37.866, E3 +425173.413}
SPL {X  -165.650, Y  +471.256, Z    +0.000, E1   -37.789, E3 +425185.066}
SPL {X  -165.650, Y  +475.981, Z    +0.000, E1   -37.909, E3 +425196.789}
SPL {X  -165.650, Y  +481.142, Z    +0.000, E1   -37.875, E3 +425210.610}
SPL {X  -165.650, Y  +487.016, Z    +0.000, E1   -37.964, E3 +425225.515}
SPL {X  -165.650, Y  +492.473, Z    +0.000, E1   -37.882, E3 +425240.311}
SPL {X  -165.650, Y  +496.967, Z    +0.000, E1   -37.731, E3 +425253.018}
SPL {X  -165.650, Y  +502.007, Z    +0.000, E1   -37.899, E3 +425265.307}
SPL {X  -165.650, Y  +507.602, Z    +0.000, E1   -37.863, E3 +425280.337}
SPL {X  -165.650, Y  +513.428, Z    +0.000, E1   -37.892, E3 +425295.403}
SPL {X  -165.650, Y  +518.534, Z    +0.000, E1   -37.976, E3 +425308.266}
SPL {X  -165.650, Y  +523.331, Z    +0.000, E1   -37.880, E3 +425321.488}
SPL {X  -165.650, Y  +528.532, Z    +0.000, E1   -37.895, E3 +425335.042}
SPL {X  -165.650, Y  +534.316, Z    +0.000, E1   -37.926, E3 +425350.156}
SPL {X  -165.650, Y  +539.968, Z    +0.000, E1   -37.796, E3 +425365.743}
SPL {X  -165.650, Y  +545.726, Z    +0.000, E1   -37.963, E3 +425379.874}
SPL {X  -165.650, Y  +550.427, Z    +0.000, E1   -37.784, E3 +425393.292}
SPL {X  -165.650, Y  +556.372, Z    +0.000, E1   -37.998, E3 +425407.688}
SPL {X  -165.650, Y  +561.478, Z    +0.000, E1   -37.846, E3 +425421.935}
SPL {X  -165.650, Y  +566.625, Z    +0.000, E1   -37.932, E3 +425434.964}
SPL {X  -165.650, Y  +571.305, Z    +0.000, E1   -37.718, E3 +425448.602}
SPL {X  -165.650, Y  +577.754, Z    +0.000, E1   -38.006, E3 +425463.893}
SPL {X  -165.650, Y  +583.042, Z    +0.000, E1   -37.879, E3 +425478.437}
SPL {X  -165.650, Y  +587.643, Z    +0.000, E1   -37.879, E3 +425490.515}
SPL {X  -165.650, Y  +592.833, Z    +0.000, E1   -37.896, E3 +425504.163}
SPL {X  -165.650, Y  +597.119, Z    +0.000, E1   -37.642, E3 +425516.892}
SPL {X  -165.650, Y  +602.808, Z    +0.000, E1   -37.983, E3 +425529.898}
SPL {X  -165.650, Y  +607.937, Z    +0.000, E1   -37.862, E3 +425544.060}
SPL {X  -165.650, Y  +612.863, Z    +0.000, E1   -37.857, E3 +425557.032}
SPL {X  -165.650, Y  +618.208, Z    +0.000, E1   -37.992, E3 +425570.275}
SPL {X  -165.650, Y  +622.884, Z    +0.000, E1   -37.770, E3 +425583.892}
SPL {X  -165.650, Y  +628.759, Z    +0.000, E1   -37.993, E3 +425598.062}
SPL {X  -165.650, Y  +633.686, Z    +0.000, E1   -37.760, E3 +425612.337}
SPL {X  -165.650, Y  +639.918, Z    +0.000, E1   -37.892, E3 +425628.145}
SPL {X  -165.650, Y  +645.851, Z    +0.000, E1   -37.854, E3 +425643.798}
SPL {X  -165.650, Y  +650.450, Z    +0.000, E1   -37.924, E3 +425655.438}
SPL {X  -165.650, Y  +654.711, Z    +0.000, E1   -37.888, E3 +425666.872}
SPL {X  -165.650, Y  +658.674, Z    +0.000, E1   -37.902, E3 +425677.140}
SPL {X  -165.650, Y  +661.754, Z    +0.000, E1   -37.878, E3 +425685.376}
SPL {X  -165.650, Y  +665.663, Z    +0.000, E1   -37.913, E3 +425695.478}
SPL {X  -165.650, Y  +669.913, Z    +0.000, E1   -37.905, E3 +425706.679}
SPL {X  -165.650, Y  +674.729, Z    +0.000, E1   -37.860, E3 +425719.689}
SPL {X  -165.591, Y  +679.928, Z    +0.000, E1   -37.818, E3 +425733.606}
SPL {X  -165.340, Y  +685.624, Z    +0.000, E1   -37.900, E3 +425748.141}
SPL {X  -165.010, Y  +690.051, Z    +0.000, E1   -37.675, E3 +425761.072}
SPL {X  -164.376, Y  +696.008, Z    +0.000, E1   -37.753, E3 +425776.436}
SPL {X  -163.617, Y  +701.375, Z    +0.000, E1   -37.486, E3 +425792.029}
SPL {X  -162.809, Y  +706.049, Z    +0.000, E1   -37.384, E3 +425804.900}
SPL {X  -161.803, Y  +710.992, Z    +0.000, E1   -37.315, E3 +425818.365}
SPL {X  -160.993, Y  +714.501, Z    +0.000, E1   -36.839, E3 +425830.241}
SPL {X  -159.156, Y  +721.427, Z    +0.000, E1   -38.526, E3 +425838.320}
SPL {X  -144.831, Y  +755.898, Z    +0.000, E1   -42.981, E3 +425899.736}
ENDSPLINE

SPLINE
SPL {X  -149.638, Y  +746.553, Z    +0.000, E1   -36.050, E3 +425984.185}
SPL {X  -161.586, Y  +711.966, Z    +0.000, E1   -22.327, E3 +425973.162}
SPL {X  -165.011, Y  +690.033, Z    +0.000, E1   -11.292, E3 +425967.546}
SPL {X  -165.581, Y  +680.273, Z    +0.000, E1    -5.775, E3 +425963.345}
SPL {X  -165.650, Y  +673.781, Z    +0.000, E1    -1.642, E3 +425962.588}
SPL {X  -165.650, Y  +669.471, Z    +0.000, E1    +1.546, E3 +425963.742}
SPL {X  -165.650, Y  +665.412, Z    +0.000, E1    +4.953, E3 +425961.768}
SPL {X  -165.650, Y  +658.891, Z    +0.000, E1   +11.031, E3 +425962.078}
SPL {X  -165.650, Y  +649.186, Z    +0.000, E1   +20.530, E3 +425963.338}
SPL {X  -165.650, Y  +637.823, Z    +0.000, E1   +39.473, E3 +425942.934}
SPL {X  -165.650, Y  +613.283, Z    +0.000, E1   +49.826, E3 +425958.501}
SPL {X  -165.650, Y  +609.693, Z    +0.000, E1   +42.113, E3 +425986.635}
SPL {X  -165.650, Y  +571.120, Z    +0.000, E1   +47.704, E3 +426031.445}
ENDSPLINE

SPLINE
SPL {X  -165.650, Y  +586.477, Z    +0.000, E1   +39.172, E3 +426047.989}
ENDSPLINE

SPLINE
SPL {X  -165.650, Y  +581.917, Z    +0.000, E1   +39.019, E3 +426060.391}
SPL {X  -165.650, Y  +577.218, Z    +0.000, E1   +38.911, E3 +426072.932}
SPL {X  -165.650, Y  +571.720, Z    +0.000, E1   +39.004, E3 +426086.323}
SPL {X  -165.650, Y  +565.656, Z    +0.000, E1   +39.042, E3 +426101.432}
SPL {X  -165.650, Y  +558.931, Z    +0.000, E1   +39.059, E3 +426118.363}
SPL {X  -165.650, Y  +552.186, Z    +0.000, E1   +39.063, E3 +426135.298}
SPL {X  -165.650, Y  +547.091, Z    +0.000, E1   +39.070, E3 +426147.958}
SPL {X  -165.650, Y  +526.098, Z    +0.000, E1   +45.792, E3 +426155.025}
SPL {X  -165.650, Y  +510.223, Z    +0.000, E1   +49.521, E3 +426162.422}
SPL {X  -165.650, Y  +506.429, Z    +0.000, E1   +48.913, E3 +426172.835}
SPL {X  -165.650, Y  +501.394, Z    +0.000, E1   +48.110, E3 +426186.814}
SPL {X  -165.650, Y  +497.138, Z    +0.000, E1   +47.280, E3 +426199.510}
SPL {X  -165.650, Y  +493.273, Z    +0.000, E1   +46.518, E3 +426211.491}
SPL {X  -165.650, Y  +489.140, Z    +0.000, E1   +45.675, E3 +426224.618}
SPL {X  -165.650, Y  +485.420, Z    +0.000, E1   +44.711, E3 +426237.837}
SPL {X  -165.650, Y  +480.756, Z    +0.000, E1   +43.779, E3 +426253.315}
SPL {X  -165.650, Y  +475.837, Z    +0.000, E1   +42.787, E3 +426269.776}
SPL {X  -165.650, Y  +472.413, Z    +0.000, E1   +41.852, E3 +426282.890}
SPL {X  -165.650, Y  +468.649, Z    +0.000, E1   +41.090, E3 +426296.254}
SPL {X  -165.650, Y  +464.675, Z    +0.000, E1   +40.045, E3 +426312.032}
SPL {X  -165.650, Y  +462.171, Z    +0.000, E1   +38.860, E3 +426325.246}
SPL {X  -165.650, Y  +457.119, Z    +0.000, E1   +39.087, E3 +426336.624}
SPL {X  -165.650, Y  +452.884, Z    +0.000, E1   +39.185, E3 +426346.672}
SPL {X  -165.650, Y  +449.593, Z    +0.000, E1   +38.852, E3 +426356.967}
SPL {X  -165.650, Y  +443.672, Z    +0.000, E1   +39.218, E3 +426369.816}
SPL {X  -165.650, Y  +436.874, Z    +0.000, E1   +39.135, E3 +426387.486}
SPL {X  -165.650, Y  +430.832, Z    +0.000, E1   +39.105, E3 +426402.674}
SPL {X  -165.650, Y  +426.072, Z    +0.000, E1   +39.194, E3 +426414.097}
SPL {X  -165.650, Y  +422.372, Z    +0.000, E1   +38.952, E3 +426424.833}
SPL {X  -165.650, Y  +417.591, Z    +0.000, E1   +39.157, E3 +426435.686}
SPL {X  -165.650, Y  +412.842, Z    +0.000, E1   +39.072, E3 +426448.185}
SPL {X  -165.650, Y  +407.612, Z    +0.000, E1   +39.068, E3 +426461.358}
SPL {X  -165.650, Y  +402.767, Z    +0.000, E1   +39.122, E3 +426473.213}
SPL {X  -165.650, Y  +398.352, Z    +0.000, E1   +39.113, E3 +426484.366}
SPL {X  -165.650, Y  +393.915, Z    +0.000, E1   +39.126, E3 +426495.443}
SPL {X  -165.650, Y  +389.523, Z    +0.000, E1   +39.115, E3 +426506.553}
SPL {X  -165.650, Y  +384.404, Z    +0.000, E1   +39.147, E3 +426519.289}
SPL {X  -165.650, Y  +378.675, Z    +0.000, E1   +39.090, E3 +426534.097}
SPL {X  -165.597, Y  +374.311, Z    +0.000, E1   +39.013, E3 +426545.383}
SPL {X  -165.438, Y  +370.129, Z    +0.000, E1   +39.090, E3 +426555.561}
SPL {X  -165.143, Y  +365.555, Z    +0.000, E1   +39.161, E3 +426566.533}
SPL {X  -164.909, Y  +362.853, Z    +0.000, E1   +38.709, E3 +426576.080}
SPL {X  -164.359, Y  +357.858, Z    +0.000, E1   +39.066, E3 +426586.542}
SPL {X  -163.818, Y  +353.935, Z    +0.000, E1   +38.811, E3 +426597.937}
SPL {X  -163.055, Y  +349.296, Z    +0.000, E1   +38.669, E3 +426610.442}
SPL {X  -162.319, Y  +345.445, Z    +0.000, E1   +38.490, E3 +426621.137}
SPL {X  -161.279, Y  +340.696, Z    +0.000, E1   +38.442, E3 +426633.465}
SPL {X  -160.251, Y  +336.552, Z    +0.000, E1   +38.166, E3 +426645.331}
SPL {X  -151.400, Y  +311.284, Z    +0.000, E1   +46.597, E3 +426653.054}
SPL {X  -146.894, Y  +301.936, Z    +0.000, E1   +40.559, E3 +426726.218}
ENDSPLINE

SPLINE
SPL {X  -154.092, Y  +317.709, Z    +0.000, E1   +32.342, E3 +426795.343}
SPL {X  -161.950, Y  +343.684, Z    +0.000, E1   +21.785, E3 +426772.182}
SPL {X  -164.623, Y  +360.087, Z    +0.000, E1   +13.426, E3 +426780.833}
SPL {X  -165.588, Y  +373.983, Z    +0.000, E1    +5.738, E3 +426773.609}
SPL {X  -165.650, Y  +380.761, Z    +0.000, E1    +1.351, E3 +426775.333}
SPL {X  -165.650, Y  +386.484, Z    +0.000, E1    -2.972, E3 +426773.340}
SPL {X  -165.650, Y  +391.786, Z    +0.000, E1    -7.566, E3 +426775.735}
SPL {X  -165.650, Y  +399.284, Z    +0.000, E1   -15.403, E3 +426770.920}
SPL {X  -165.650, Y  +409.824, Z    +0.000, E1   -26.455, E3 +426768.800}
SPL {X  -165.650, Y  +437.337, Z    +0.000, E1   -46.817, E3 +426771.435}
SPL {X  -165.650, Y  +450.640, Z    +0.000, E1   -46.274, E3 +426793.457}
SPL {X  -165.650, Y  +484.108, Z    +0.000, E1   -48.531, E3 +426838.236}
ENDSPLINE

SPLINE
SPL {X  -165.650, Y  +465.194, Z    +0.000, E1   -39.630, E3 +426850.104}
ENDSPLINE

SPLINE
SPL {X  -165.650, Y  +465.900, Z    +0.000, E1   -37.888, E3 +426862.807}
SPL {X  -165.650, Y  +471.256, Z    +0.000, E1   -37.789, E3 +426877.374}
SPL {X  -165.650, Y  +475.981, Z    +0.000, E1   -37.909, E3 +426889.097}
SPL {X  -165.650, Y  +481.142, Z    +0.000, E1   -37.875, E3 +426902.917}
SPL {X  -165.650, Y  +487.016, Z    +0.000, E1   -37.964, E3 +426917.823}
SPL {X  -165.650, Y  +492.473, Z    +0.000, E1   -37.882, E3 +426932.619}
SPL {X  -165.650, Y  +496.967, Z    +0.000, E1   -37.731, E3 +426945.326}
SPL {X  -165.650, Y  +502.007, Z    +0.000, E1   -37.899, E3 +426957.615}
SPL {X  -165.650, Y  +506.838, Z    +0.000, E1   -38.018, E3 +426969.512}
SPL {X  -165.650, Y  +512.106, Z    +0.000, E1   -37.811, E3 +426984.854}
SPL {X  -165.650, Y  +518.534, Z    +0.000, E1   -37.976, E3 +427000.574}
SPL {X  -165.650, Y  +523.331, Z    +0.000, E1   -37.880, E3 +427013.796}
SPL {X  -165.650, Y  +528.532, Z    +0.000, E1   -37.895, E3 +427027.349}
SPL {X  -165.650, Y  +532.864, Z    +0.000, E1   -37.846, E3 +427038.991}
SPL {X  -165.650, Y  +537.279, Z    +0.000, E1   -37.980, E3 +427049.813}
SPL {X  -165.650, Y  +542.501, Z    +0.000, E1   -37.886, E3 +427064.157}
SPL {X  -165.650, Y  +546.598, Z    +0.000, E1   -37.767, E3 +427075.509}
SPL {X  -165.650, Y  +550.427, Z    +0.000, E1   -37.784, E3 +427085.599}
SPL {X  -165.650, Y  +554.659, Z    +0.000, E1   -37.927, E3 +427095.783}
SPL {X  -165.650, Y  +557.856, Z    +0.000, E1   -37.998, E3 +427103.733}
SPL {X  -165.650, Y  +561.478, Z    +0.000, E1   -37.846, E3 +427114.243}
SPL {X  -165.650, Y  +566.625, Z    +0.000, E1   -37.932, E3 +427127.272}
SPL {X  -165.650, Y  +571.305, Z    +0.000, E1   -37.718, E3 +427140.909}
SPL {X  -165.650, Y  +577.754, Z    +0.000, E1   -38.006, E3 +427156.201}
SPL {X  -165.650, Y  +583.042, Z    +0.000, E1   -37.879, E3 +427170.744}
SPL {X  -165.650, Y  +587.643, Z    +0.000, E1   -37.879, E3 +427182.822}
SPL {X  -165.650, Y  +592.833, Z    +0.000, E1   -37.896, E3 +427196.471}
SPL {X  -165.650, Y  +597.119, Z    +0.000, E1   -37.642, E3 +427209.200}
SPL {X  -165.650, Y  +602.808, Z    +0.000, E1   -37.983, E3 +427222.206}
SPL {X  -165.650, Y  +607.937, Z    +0.000, E1   -37.862, E3 +427236.367}
SPL {X  -165.650, Y  +614.056, Z    +0.000, E1   -37.933, E3 +427252.138}
SPL {X  -165.650, Y  +619.142, Z    +0.000, E1   -37.954, E3 +427265.157}
SPL {X  -165.650, Y  +622.884, Z    +0.000, E1   -37.770, E3 +427276.200}
SPL {X  -165.650, Y  +628.759, Z    +0.000, E1   -37.993, E3 +427290.369}
SPL {X  -165.650, Y  +633.686, Z    +0.000, E1   -37.760, E3 +427304.645}
SPL {X  -165.650, Y  +638.669, Z    +0.000, E1   -37.941, E3 +427316.651}
SPL {X  -165.650, Y  +643.208, Z    +0.000, E1   -37.786, E3 +427329.568}
SPL {X  -165.650, Y  +649.293, Z    +0.000, E1   -37.920, E3 +427344.858}
SPL {X  -165.650, Y  +654.711, Z    +0.000, E1   -37.888, E3 +427359.180}
SPL {X  -165.650, Y  +660.285, Z    +0.000, E1   -37.928, E3 +427373.698}
SPL {X  -165.650, Y  +665.663, Z    +0.000, E1   -37.913, E3 +427387.785}
SPL {X  -165.650, Y  +671.321, Z    +0.000, E1   -37.904, E3 +427402.887}
SPL {X  -165.649, Y  +676.172, Z    +0.000, E1   -37.873, E3 +427415.583}
SPL {X  -165.554, Y  +681.132, Z    +0.000, E1   -37.883, E3 +427428.831}
SPL {X  -165.277, Y  +686.615, Z    +0.000, E1   -37.853, E3 +427443.213}
SPL {X  -164.889, Y  +691.361, Z    +0.000, E1   -37.742, E3 +427456.567}
SPL {X  -164.246, Y  +697.018, Z    +0.000, E1   -37.690, E3 +427471.609}
SPL {X  -163.617, Y  +701.375, Z    +0.000, E1   -37.486, E3 +427484.336}
SPL {X  -162.809, Y  +706.049, Z    +0.000, E1   -37.384, E3 +427497.208}
SPL {X  -161.803, Y  +710.992, Z    +0.000, E1   -37.315, E3 +427510.672}
SPL {X  -160.993, Y  +714.501, Z    +0.000, E1   -36.839, E3 +427522.549}
SPL {X  -159.156, Y  +721.427, Z    +0.000, E1   -38.526, E3 +427530.627}
SPL {X  -144.831, Y  +755.898, Z    +0.000, E1   -42.981, E3 +427592.043}
ENDSPLINE

SPLINE
SPL {X  -153.047, Y  +738.876, Z    +0.000, E1   -33.363, E3 +427674.258}
SPL {X  -162.649, Y  +706.888, Z    +0.000, E1   -19.911, E3 +427663.620}
SPL {X  -165.011, Y  +690.033, Z    +0.000, E1   -11.292, E3 +427659.854}
SPL {X  -165.581, Y  +680.273, Z    +0.000, E1    -5.775, E3 +427655.652}
SPL {X  -165.650, Y  +673.781, Z    +0.000, E1    -1.642, E3 +427654.896}
SPL {X  -165.650, Y  +669.471, Z    +0.000, E1    +1.546, E3 +427656.050}
SPL {X  -165.650, Y  +665.412, Z    +0.000, E1    +4.953, E3 +427654.075}
SPL {X  -165.650, Y  +658.891, Z    +0.000, E1   +11.031, E3 +427654.386}
SPL {X  -165.650, Y  +649.186, Z    +0.000, E1   +20.530, E3 +427655.646}
SPL {X  -165.650, Y  +637.823, Z    +0.000, E1   +39.473, E3 +427635.242}
SPL {X  -165.650, Y  +614.460, Z    +0.000, E1   +51.116, E3 +427646.110}
SPL {X  -165.650, Y  +609.746, Z    +0.000, E1   +42.762, E3 +427676.768}
SPL {X  -165.650, Y  +571.120, Z    +0.000, E1   +47.704, E3 +427723.752}
ENDSPLINE

SPLINE
SPL {X  -165.650, Y  +586.477, Z    +0.000, E1   +39.172, E3 +427740.297}
ENDSPLINE

SPLINE
SPL {X  -165.650, Y  +581.917, Z    +0.000, E1   +39.019, E3 +427752.699}
SPL {X  -165.650, Y  +577.218, Z    +0.000, E1   +38.911, E3 +427765.239}
SPL {X  -165.650, Y  +572.890, Z    +0.000, E1   +39.033, E3 +427775.377}
SPL {X  -165.650, Y  +569.005, Z    +0.000, E1   +38.999, E3 +427785.468}
SPL {X  -165.650, Y  +564.604, Z    +0.000, E1   +38.986, E3 +427796.603}
SPL {X  -165.650, Y  +558.931, Z    +0.000, E1   +39.059, E3 +427810.671}
SPL {X  -165.650, Y  +553.380, Z    +0.000, E1   +39.004, E3 +427824.834}
SPL {X  -165.650, Y  +548.147, Z    +0.000, E1   +39.104, E3 +427837.514}
SPL {X  -165.650, Y  +526.098, Z    +0.000, E1   +45.792, E3 +427847.332}
SPL {X  -165.650, Y  +510.223, Z    +0.000, E1   +49.521, E3 +427854.730}
SPL {X  -165.650, Y  +506.429, Z    +0.000, E1   +48.913, E3 +427865.143}
SPL {X  -165.650, Y  +501.394, Z    +0.000, E1   +48.110, E3 +427879.122}
SPL {X  -165.650, Y  +497.138, Z    +0.000, E1   +47.280, E3 +427891.818}
SPL {X  -165.650, Y  +493.273, Z    +0.000, E1   +46.518, E3 +427903.799}
SPL {X  -165.650, Y  +489.140, Z    +0.000, E1   +45.675, E3 +427916.926}
SPL {X  -165.650, Y  +485.420, Z    +0.000, E1   +44.711, E3 +427930.145}
SPL {X  -165.650, Y  +482.261, Z    +0.000, E1   +43.960, E3 +427941.097}
SPL {X  -165.650, Y  +478.467, Z    +0.000, E1   +43.371, E3 +427952.924}
SPL {X  -165.650, Y  +474.990, Z    +0.000, E1   +42.535, E3 +427965.276}
SPL {X  -165.650, Y  +471.308, Z    +0.000, E1   +41.710, E3 +427978.782}
SPL {X  -165.650, Y  +467.130, Z    +0.000, E1   +40.624, E3 +427994.907}
SPL {X  -165.650, Y  +463.869, Z    +0.000, E1   +39.839, E3 +428007.375}
SPL {X  -165.650, Y  +462.171, Z    +0.000, E1   +38.860, E3 +428017.554}
SPL {X  -165.650, Y  +457.119, Z    +0.000, E1   +39.087, E3 +428028.932}
SPL {X  -165.650, Y  +452.884, Z    +0.000, E1   +39.185, E3 +428038.980}
SPL {X  -165.650, Y  +449.593, Z    +0.000, E1   +38.852, E3 +428049.274}
SPL {X  -165.650, Y  +445.147, Z    +0.000, E1   +39.088, E3 +428059.097}
SPL {X  -165.650, Y  +439.751, Z    +0.000, E1   +39.254, E3 +428071.714}
SPL {X  -165.650, Y  +435.510, Z    +0.000, E1   +39.051, E3 +428083.525}
SPL {X  -165.650, Y  +430.832, Z    +0.000, E1   +39.105, E3 +428094.982}
SPL {X  -165.650, Y  +426.072, Z    +0.000, E1   +39.194, E3 +428106.405}
SPL {X  -165.650, Y  +422.372, Z    +0.000, E1   +38.952, E3 +428117.141}
SPL {X  -165.650, Y  +417.591, Z    +0.000, E1   +39.157, E3 +428127.994}
SPL {X  -165.650, Y  +412.842, Z    +0.000, E1   +39.072, E3 +428140.492}
SPL {X  -165.650, Y  +407.612, Z    +0.000, E1   +39.068, E3 +428153.665}
SPL {X  -165.650, Y  +402.767, Z    +0.000, E1   +39.122, E3 +428165.521}
SPL {X  -165.650, Y  +398.352, Z    +0.000, E1   +39.113, E3 +428176.674}
SPL {X  -165.650, Y  +393.915, Z    +0.000, E1   +39.126, E3 +428187.751}
SPL {X  -165.650, Y  +389.523, Z    +0.000, E1   +39.115, E3 +428198.861}
SPL {X  -165.650, Y  +384.404, Z    +0.000, E1   +39.147, E3 +428211.596}
SPL {X  -165.650, Y  +380.058, Z    +0.000, E1   +39.073, E3 +428222.884}
SPL {X  -165.624, Y  +375.547, Z    +0.000, E1   +39.047, E3 +428234.483}
SPL {X  -165.438, Y  +370.129, Z    +0.000, E1   +39.090, E3 +428247.868}
SPL {X  -165.143, Y  +365.555, Z    +0.000, E1   +39.161, E3 +428258.841}
SPL {X  -164.909, Y  +362.853, Z    +0.000, E1   +38.709, E3 +428268.387}
SPL {X  -164.359, Y  +357.858, Z    +0.000, E1   +39.066, E3 +428278.850}
SPL {X  -163.818, Y  +353.935, Z    +0.000, E1   +38.811, E3 +428290.244}
SPL {X  -163.055, Y  +349.296, Z    +0.000, E1   +38.669, E3 +428302.750}
SPL {X  -162.021, Y  +344.016, Z    +0.000, E1   +38.517, E3 +428317.039}
SPL {X  -160.588, Y  +337.861, Z    +0.000, E1   +38.304, E3 +428333.753}
SPL {X  -153.716, Y  +316.763, Z    +0.000, E1   +45.637, E3 +428340.257}
SPL {X  -149.011, Y  +306.142, Z    +0.000, E1   +47.422, E3 +428350.288}
SPL {X  -146.894, Y  +301.936, Z    +0.000, E1   +40.559, E3 +428418.526}
ENDSPLINE

SPLINE
SPL {X  -154.092, Y  +317.709, Z    +0.000, E1   +32.342, E3 +428487.650}
SPL {X  -161.950, Y  +343.684, Z    +0.000, E1   +21.785, E3 +428464.490}
SPL {X  -164.623, Y  +360.087, Z    +0.000, E1   +13.426, E3 +428473.140}
SPL {X  -165.489, Y  +371.187, Z    +0.000, E1    +7.370, E3 +428463.981}
SPL {X  -165.621, Y  +375.403, Z    +0.000, E1    +4.810, E3 +428466.879}
SPL {X  -165.650, Y  +380.761, Z    +0.000, E1    +1.351, E3 +428467.641}
SPL {X  -165.650, Y  +386.484, Z    +0.000, E1    -2.972, E3 +428465.648}
SPL {X  -165.650, Y  +392.905, Z    +0.000, E1    -8.557, E3 +428467.702}
SPL {X  -165.650, Y  +404.146, Z    +0.000, E1   -20.514, E3 +428462.432}
SPL {X  -165.650, Y  +416.920, Z    +0.000, E1   -34.832, E3 +428456.395}
SPL {X  -165.650, Y  +445.455, Z    +0.000, E1   -46.044, E3 +428478.486}
SPL {X  -165.650, Y  +459.839, Z    +0.000, E1   -48.128, E3 +428493.552}
SPL {X  -165.650, Y  +484.108, Z    +0.000, E1   -48.531, E3 +428530.544}
ENDSPLINE

SPLINE
SPL {X  -165.650, Y  +464.452, Z    +0.000, E1   -38.833, E3 +428545.604}
ENDSPLINE

SPLINE
SPL {X  -165.650, Y  +467.011, Z    +0.000, E1   -37.866, E3 +428558.028}
SPL {X  -165.650, Y  +471.256, Z    +0.000, E1   -37.789, E3 +428569.682}
SPL {X  -165.650, Y  +475.981, Z    +0.000, E1   -37.909, E3 +428581.405}
SPL {X  -165.650, Y  +481.142, Z    +0.000, E1   -37.875, E3 +428595.225}
SPL {X  -165.650, Y  +487.016, Z    +0.000, E1   -37.964, E3 +428610.130}
SPL {X  -165.650, Y  +492.473, Z    +0.000, E1   -37.882, E3 +428624.927}
SPL {X  -165.650, Y  +496.967, Z    +0.000, E1   -37.731, E3 +428637.634}
SPL {X  -165.650, Y  +502.007, Z    +0.000, E1   -37.899, E3 +428649.923}
SPL {X  -165.650, Y  +506.838, Z    +0.000, E1   -38.018, E3 +428661.820}
SPL {X  -165.650, Y  +510.962, Z    +0.000, E1   -37.876, E3 +428673.534}
SPL {X  -165.650, Y  +516.973, Z    +0.000, E1   -37.871, E3 +428689.560}
SPL {X  -165.650, Y  +523.331, Z    +0.000, E1   -37.880, E3 +428706.103}
SPL {X  -165.650, Y  +528.532, Z    +0.000, E1   -37.895, E3 +428719.657}
SPL {X  -165.650, Y  +532.864, Z    +0.000, E1   -37.846, E3 +428731.299}
SPL {X  -165.650, Y  +537.279, Z    +0.000, E1   -37.980, E3 +428742.121}
SPL {X  -165.650, Y  +542.501, Z    +0.000, E1   -37.886, E3 +428756.464}
SPL {X  -165.650, Y  +546.598, Z    +0.000, E1   -37.767, E3 +428767.817}
SPL {X  -165.650, Y  +550.427, Z    +0.000, E1   -37.784, E3 +428777.907}
SPL {X  -165.650, Y  +556.372, Z    +0.000, E1   -37.998, E3 +428792.303}
SPL {X  -165.650, Y  +561.478, Z    +0.000, E1   -37.846, E3 +428806.550}
SPL {X  -165.650, Y  +566.625, Z    +0.000, E1   -37.932, E3 +428819.580}
SPL {X  -165.650, Y  +571.305, Z    +0.000, E1   -37.718, E3 +428833.217}
SPL {X  -165.650, Y  +576.676, Z    +0.000, E1   -38.057, E3 +428845.213}
SPL {X  -165.650, Y  +581.909, Z    +0.000, E1   -37.903, E3 +428860.085}
SPL {X  -165.650, Y  +587.643, Z    +0.000, E1   -37.879, E3 +428875.130}
SPL {X  -165.650, Y  +592.833, Z    +0.000, E1   -37.896, E3 +428888.779}
SPL {X  -165.650, Y  +599.187, Z    +0.000, E1   -37.841, E3 +428905.917}
SPL {X  -165.650, Y  +604.276, Z    +0.000, E1   -37.917, E3 +428918.604}
SPL {X  -165.650, Y  +607.937, Z    +0.000, E1   -37.862, E3 +428928.675}
SPL {X  -165.650, Y  +612.863, Z    +0.000, E1   -37.857, E3 +428941.648}
SPL {X  -165.650, Y  +618.208, Z    +0.000, E1   -37.992, E3 +428954.890}
SPL {X  -165.650, Y  +622.884, Z    +0.000, E1   -37.770, E3 +428968.507}
SPL {X  -165.650, Y  +627.016, Z    +0.000, E1   -37.897, E3 +428978.546}
SPL {X  -165.650, Y  +630.421, Z    +0.000, E1   -38.020, E3 +428986.708}
SPL {X  -165.650, Y  +633.686, Z    +0.000, E1   -37.760, E3 +428996.952}
SPL {X  -165.650, Y  +638.669, Z    +0.000, E1   -37.941, E3 +429008.959}
SPL {X  -165.650, Y  +643.208, Z    +0.000, E1   -37.786, E3 +429021.875}
SPL {X  -165.650, Y  +649.293, Z    +0.000, E1   -37.920, E3 +429037.165}
SPL {X  -165.650, Y  +654.711, Z    +0.000, E1   -37.888, E3 +429051.487}
SPL {X  -165.650, Y  +658.674, Z    +0.000, E1   -37.902, E3 +429061.755}
SPL {X  -165.650, Y  +661.754, Z    +0.000, E1   -37.878, E3 +429069.991}
SPL {X  -165.650, Y  +665.663, Z    +0.000, E1   -37.913, E3 +429080.093}
SPL {X  -165.650, Y  +671.321, Z    +0.000, E1   -37.904, E3 +429095.194}
SPL {X  -165.649, Y  +676.172, Z    +0.000, E1   -37.873, E3 +429107.891}
SPL {X  -165.591, Y  +679.928, Z    +0.000, E1   -37.818, E3 +429118.222}
SPL {X  -165.340, Y  +685.624, Z    +0.000, E1   -37.900, E3 +429132.756}
SPL {X  -165.010, Y  +690.051, Z    +0.000, E1   -37.675, E3 +429145.687}
SPL {X  -164.652, Y  +693.652, Z    +0.000, E1   -37.750, E3 +429154.617}
SPL {X  -164.143, Y  +697.797, Z    +0.000, E1   -37.636, E3 +429166.437}
SPL {X  -163.447, Y  +702.423, Z    +0.000, E1   -37.496, E3 +429179.245}
SPL {X  -162.809, Y  +706.049, Z    +0.000, E1   -37.384, E3 +429189.516}
SPL {X  -162.124, Y  +709.497, Z    +0.000, E1   -37.325, E3 +429198.838}
SPL {X  -161.242, Y  +713.462, Z    +0.000, E1   -37.074, E3 +429210.959}
SPL {X  -159.156, Y  +721.427, Z    +0.000, E1   -38.526, E3 +429222.935}
SPL {X  -144.831, Y  +755.898, Z    +0.000, E1   -42.981, E3 +429284.351}
ENDSPLINE

SPLINE
SPL {X  -153.047, Y  +738.876, Z    +0.000, E1   -33.363, E3 +429366.566}
SPL {X  -162.649, Y  +706.888, Z    +0.000, E1   -19.911, E3 +429355.927}
SPL {X  -165.011, Y  +690.033, Z    +0.000, E1   -11.292, E3 +429352.162}
SPL {X  -165.581, Y  +680.273, Z    +0.000, E1    -5.775, E3 +429347.960}
SPL {X  -165.650, Y  +674.660, Z    +0.000, E1    -2.196, E3 +429348.627}
SPL {X  -165.650, Y  +669.932, Z    +0.000, E1    +1.173, E3 +429347.203}
SPL {X  -165.650, Y  +665.412, Z    +0.000, E1    +4.953, E3 +429346.383}
SPL {X  -165.650, Y  +660.335, Z    +0.000, E1    +9.682, E3 +429346.900}
SPL {X  -165.650, Y  +650.970, Z    +0.000, E1   +18.783, E3 +429347.448}
SPL {X  -165.650, Y  +637.823, Z    +0.000, E1   +39.473, E3 +429327.550}
SPL {X  -165.650, Y  +614.460, Z    +0.000, E1   +51.116, E3 +429338.418}
SPL {X  -165.650, Y  +609.746, Z    +0.000, E1   +42.762, E3 +429369.076}
SPL {X  -165.650, Y  +571.120, Z    +0.000, E1   +47.704, E3 +429416.060}
ENDSPLINE

SPLINE
SPL {X  -165.650, Y  +586.477, Z    +0.000, E1   +39.172, E3 +429432.604}
ENDSPLINE

SPLINE
SPL {X  -165.650, Y  +581.917, Z    +0.000, E1   +39.019, E3 +429445.007}
SPL {X  -165.650, Y  +577.218, Z    +0.000, E1   +38.911, E3 +429457.547}
SPL {X  -165.650, Y  +572.890, Z    +0.000, E1   +39.033, E3 +429467.685}
SPL {X  -165.650, Y  +569.005, Z    +0.000, E1   +38.999, E3 +429477.775}
SPL {X  -165.650, Y  +564.604, Z    +0.000, E1   +38.986, E3 +429488.911}
SPL {X  -165.650, Y  +558.931, Z    +0.000, E1   +39.059, E3 +429502.979}
SPL {X  -165.650, Y  +553.380, Z    +0.000, E1   +39.004, E3 +429517.142}
SPL {X  -165.650, Y  +548.147, Z    +0.000, E1   +39.104, E3 +429529.821}
SPL {X  -165.650, Y  +526.098, Z    +0.000, E1   +45.792, E3 +429539.640}
SPL {X  -165.650, Y  +510.223, Z    +0.000, E1   +49.521, E3 +429547.037}
SPL {X  -165.650, Y  +506.429, Z    +0.000, E1   +48.913, E3 +429557.450}
SPL {X  -165.650, Y  +501.394, Z    +0.000, E1   +48.110, E3 +429571.429}
SPL {X  -165.650, Y  +497.138, Z    +0.000, E1   +47.280, E3 +429584.125}
SPL {X  -165.650, Y  +493.273, Z    +0.000, E1   +46.518, E3 +429596.106}
SPL {X  -165.650, Y  +489.140, Z    +0.000, E1   +45.675, E3 +429609.234}
SPL {X  -165.650, Y  +485.420, Z    +0.000, E1   +44.711, E3 +429622.453}
SPL {X  -165.650, Y  +480.756, Z    +0.000, E1   +43.779, E3 +429637.931}
SPL {X  -165.650, Y  +475.837, Z    +0.000, E1   +42.787, E3 +429654.391}
SPL {X  -165.650, Y  +472.413, Z    +0.000, E1   +41.852, E3 +429667.506}
SPL {X  -165.650, Y  +468.649, Z    +0.000, E1   +41.090, E3 +429680.869}
SPL {X  -165.650, Y  +464.675, Z    +0.000, E1   +40.045, E3 +429696.647}
SPL {X  -165.650, Y  +462.171, Z    +0.000, E1   +38.860, E3 +429709.861}
SPL {X  -165.650, Y  +457.119, Z    +0.000, E1   +39.087, E3 +429721.240}
SPL {X  -165.650, Y  +452.884, Z    +0.000, E1   +39.185, E3 +429731.287}
SPL {X  -165.650, Y  +449.593, Z    +0.000, E1   +38.852, E3 +429741.582}
SPL {X  -165.650, Y  +445.147, Z    +0.000, E1   +39.088, E3 +429751.404}
SPL {X  -165.650, Y  +439.751, Z    +0.000, E1   +39.254, E3 +429764.022}
SPL {X  -165.650, Y  +435.510, Z    +0.000, E1   +39.051, E3 +429775.833}
SPL {X  -165.650, Y  +430.832, Z    +0.000, E1   +39.105, E3 +429787.290}
SPL {X  -165.650, Y  +426.072, Z    +0.000, E1   +39.194, E3 +429798.713}
SPL {X  -165.650, Y  +422.372, Z    +0.000, E1   +38.952, E3 +429809.448}
SPL {X  -165.650, Y  +417.591, Z    +0.000, E1   +39.157, E3 +429820.301}
SPL {X  -165.650, Y  +412.842, Z    +0.000, E1   +39.072, E3 +429832.800}
SPL {X  -165.650, Y  +407.612, Z    +0.000, E1   +39.068, E3 +429845.973}
SPL {X  -165.650, Y  +402.767, Z    +0.000, E1   +39.122, E3 +429857.828}
SPL {X  -165.650, Y  +398.352, Z    +0.000, E1   +39.113, E3 +429868.981}
SPL {X  -165.650, Y  +393.915, Z    +0.000, E1   +39.126, E3 +429880.058}
SPL {X  -165.650, Y  +388.386, Z    +0.000, E1   +39.140, E3 +429894.008}
SPL {X  -165.650, Y  +383.342, Z    +0.000, E1   +39.144, E3 +429906.495}
SPL {X  -165.650, Y  +378.675, Z    +0.000, E1   +39.090, E3 +429918.712}
SPL {X  -165.597, Y  +374.311, Z    +0.000, E1   +39.013, E3 +429929.998}
SPL {X  -165.438, Y  +370.129, Z    +0.000, E1   +39.090, E3 +429940.176}
SPL {X  -165.143, Y  +365.555, Z    +0.000, E1   +39.161, E3 +429951.148}
SPL {X  -164.909, Y  +362.853, Z    +0.000, E1   +38.709, E3 +429960.695}
SPL {X  -164.359, Y  +357.858, Z    +0.000, E1   +39.066, E3 +429971.158}
SPL {X  -163.818, Y  +353.935, Z    +0.000, E1   +38.811, E3 +429982.552}
SPL {X  -163.055, Y  +349.296, Z    +0.000, E1   +38.669, E3 +429995.057}
SPL {X  -162.319, Y  +345.445, Z    +0.000, E1   +38.490, E3 +430005.753}
SPL {X  -161.279, Y  +340.696, Z    +0.000, E1   +38.442, E3 +430018.080}
SPL {X  -160.251, Y  +336.552, Z    +0.000, E1   +38.166, E3 +430029.946}
SPL {X  -151.400, Y  +311.284, Z    +0.000, E1   +46.597, E3 +430037.669}
SPL {X  -146.894, Y  +301.936, Z    +0.000, E1   +40.559, E3 +430110.834}
ENDSPLINE

SPLINE
SPL {X  -154.092, Y  +317.709, Z    +0.000, E1   +32.342, E3 +430179.958}
SPL {X  -161.950, Y  +343.684, Z    +0.000, E1   +21.785, E3 +430156.797}
SPL {X  -164.623, Y  +360.087, Z    +0.000, E1   +13.426, E3 +430165.448}
SPL {X  -165.489, Y  +371.187, Z    +0.000, E1    +7.370, E3 +430156.289}
SPL {X  -165.621, Y  +375.403, Z    +0.000, E1    +4.810, E3 +430159.187}
SPL {X  -165.650, Y  +380.761, Z    +0.000, E1    +1.351, E3 +430159.949}
SPL {X  -165.650, Y  +386.484, Z    +0.000, E1    -2.972, E3 +430157.956}
SPL {X  -165.650, Y  +392.905, Z    +0.000, E1    -8.557, E3 +430160.010}
SPL {X  -165.650, Y  +404.146, Z    +0.000, E1   -20.514, E3 +430154.740}
SPL {X  -165.650, Y  +412.709, Z    +0.000, E1   -30.621, E3 +430149.703}
SPL {X  -165.650, Y  +437.337, Z    +0.000, E1   -46.817, E3 +430156.051}
SPL {X  -165.650, Y  +450.640, Z    +0.000, E1   -46.274, E3 +430178.073}
SPL {X  -165.650, Y  +484.108, Z    +0.000, E1   -48.531, E3 +430222.851}
ENDSPLINE

SPLINE
SPL {X  -165.650, Y  +464.452, Z    +0.000, E1   -38.833, E3 +430237.912}
ENDSPLINE

SPLINE
SPL {X  -165.650, Y  +467.011, Z    +0.000, E1   -37.866, E3 +430250.336}
SPL {X  -165.650, Y  +471.256, Z    +0.000, E1   -37.789, E3 +430261.989}
SPL {X  -165.650, Y  +475.981, Z    +0.000, E1   -37.909, E3 +430273.712}
SPL {X  -165.650, Y  +481.142, Z    +0.000, E1   -37.875, E3 +430287.533}
SPL {X  -165.650, Y  +487.016, Z    +0.000, E1   -37.964, E3 +430302.438}
SPL {X  -165.650, Y  +492.473, Z    +0.000, E1   -37.882, E3 +430317.234}
SPL {X  -165.650, Y  +496.967, Z    +0.000, E1   -37.731, E3 +430329.941}
SPL {X  -165.650, Y  +502.007, Z    +0.000, E1   -37.899, E3 +430342.230}
SPL {X  -165.650, Y  +507.602, Z    +0.000, E1   -37.863, E3 +430357.260}
SPL {X  -165.650, Y  +513.428, Z    +0.000, E1   -37.892, E3 +430372.326}
SPL {X  -165.650, Y  +518.534, Z    +0.000, E1   -37.976, E3 +430385.190}
SPL {X  -165.650, Y  +523.331, Z    +0.000, E1   -37.880, E3 +430398.411}
SPL {X  -165.650, Y  +528.532, Z    +0.000, E1   -37.895, E3 +430411.965}
SPL {X  -165.650, Y  +532.864, Z    +0.000, E1   -37.846, E3 +430423.606}
SPL {X  -165.650, Y  +537.279, Z    +0.000, E1   -37.980, E3 +430434.429}
SPL {X  -165.650, Y  +540.651, Z    +0.000, E1   -37.651, E3 +430445.231}
SPL {X  -165.650, Y  +545.726, Z    +0.000, E1   -37.963, E3 +430456.797}
SPL {X  -165.650, Y  +550.427, Z    +0.000, E1   -37.784, E3 +430470.215}
SPL {X  -165.650, Y  +554.659, Z    +0.000, E1   -37.927, E3 +430480.399}
SPL {X  -165.650, Y  +557.856, Z    +0.000, E1   -37.998, E3 +430488.349}
SPL {X  -165.650, Y  +562.748, Z    +0.000, E1   -37.890, E3 +430502.091}
SPL {X  -165.650, Y  +567.848, Z    +0.000, E1   -37.954, E3 +430514.864}
SPL {X  -165.650, Y  +571.305, Z    +0.000, E1   -37.718, E3 +430525.525}
SPL {X  -165.650, Y  +577.754, Z    +0.000, E1   -38.006, E3 +430540.816}
SPL {X  -165.650, Y  +583.042, Z    +0.000, E1   -37.879, E3 +430555.360}
SPL {X  -165.650, Y  +587.643, Z    +0.000, E1   -37.879, E3 +430567.438}
SPL {X  -165.650, Y  +592.833, Z    +0.000, E1   -37.896, E3 +430581.086}
SPL {X  -165.650, Y  +599.187, Z    +0.000, E1   -37.841, E3 +430598.224}
SPL {X  -165.650, Y  +604.276, Z    +0.000, E1   -37.917, E3 +430610.912}
SPL {X  -165.650, Y  +607.937, Z    +0.000, E1   -37.862, E3 +430620.983}
SPL {X  -165.650, Y  +612.863, Z    +0.000, E1   -37.857, E3 +430633.955}
SPL {X  -165.650, Y  +618.208, Z    +0.000, E1   -37.992, E3 +430647.198}
SPL {X  -165.650, Y  +622.884, Z    +0.000, E1   -37.770, E3 +430660.815}
SPL {X  -165.650, Y  +628.759, Z    +0.000, E1   -37.993, E3 +430674.985}
SPL {X  -165.650, Y  +633.686, Z    +0.000, E1   -37.760, E3 +430689.260}
SPL {X  -165.650, Y  +638.669, Z    +0.000, E1   -37.941, E3 +430701.267}
SPL {X  -165.650, Y  +644.441, Z    +0.000, E1   -37.838, E3 +430717.282}
SPL {X  -165.650, Y  +650.450, Z    +0.000, E1   -37.924, E3 +430732.361}
SPL {X  -165.650, Y  +654.711, Z    +0.000, E1   -37.888, E3 +430743.795}
SPL {X  -165.650, Y  +660.285, Z    +0.000, E1   -37.928, E3 +430758.313}
SPL {X  -165.650, Y  +665.663, Z    +0.000, E1   -37.913, E3 +430772.401}
SPL {X  -165.650, Y  +669.913, Z    +0.000, E1   -37.905, E3 +430783.602}
SPL {X  -165.650, Y  +674.729, Z    +0.000, E1   -37.860, E3 +430796.612}
SPL {X  -165.554, Y  +681.132, Z    +0.000, E1   -37.883, E3 +430813.446}
SPL {X  -165.277, Y  +686.615, Z    +0.000, E1   -37.853, E3 +430827.828}
SPL {X  -164.889, Y  +691.361, Z    +0.000, E1   -37.742, E3 +430841.182}
SPL {X  -164.246, Y  +697.018, Z    +0.000, E1   -37.690, E3 +430856.224}
SPL {X  -163.617, Y  +701.375, Z    +0.000, E1   -37.486, E3 +430868.952}
SPL {X  -162.809, Y  +706.049, Z    +0.000, E1   -37.384, E3 +430881.823}
SPL {X  -161.803, Y  +710.992, Z    +0.000, E1   -37.315, E3 +430895.288}
SPL {X  -160.993, Y  +714.501, Z    +0.000, E1   -36.839, E3 +430907.164}
SPL {X  -159.156, Y  +721.427, Z    +0.000, E1   -38.526, E3 +430915.243}
SPL {X  -144.831, Y  +755.898, Z    +0.000, E1   -42.981, E3 +430976.659}
ENDSPLINE

SPLINE
SPL {X  -149.638, Y  +746.553, Z    +0.000, E1   -36.050, E3 +431061.108}
SPL {X  -161.586, Y  +711.966, Z    +0.000, E1   -22.327, E3 +431050.086}
SPL {X  -165.011, Y  +690.033, Z    +0.000, E1   -11.292, E3 +431044.469}
SPL {X  -165.581, Y  +680.273, Z    +0.000, E1    -5.775, E3 +431040.268}
SPL {X  -165.650, Y  +673.781, Z    +0.000, E1    -1.642, E3 +431039.511}
SPL {X  -165.650, Y  +669.471, Z    +0.000, E1    +1.546, E3 +431040.666}
SPL {X  -165.650, Y  +665.412, Z    +0.000, E1    +4.953, E3 +431038.691}
SPL {X  -165.650, Y  +658.891, Z    +0.000, E1   +11.031, E3 +431039.001}
SPL {X  -165.650, Y  +649.186, Z    +0.000, E1   +20.530, E3 +431040.261}
SPL {X  -165.650, Y  +637.823, Z    +0.000, E1   +39.473, E3 +431019.857}
SPL {X  -165.650, Y  +613.283, Z    +0.000, E1   +49.826, E3 +431035.424}
SPL {X  -165.650, Y  +609.693, Z    +0.000, E1   +42.113, E3 +431063.559}
SPL {X  -165.650, Y  +571.120, Z    +0.000, E1   +47.704, E3 +431108.368}
ENDSPLINE

SPLINE
SPL {X  -165.650, Y  +586.477, Z    +0.000, E1   +39.172, E3 +431124.912}
ENDSPLINE

SPLINE
SPL {X  -165.650, Y  +581.917, Z    +0.000, E1   +39.019, E3 +431137.314}
SPL {X  -165.650, Y  +577.218, Z    +0.000, E1   +38.911, E3 +431149.855}
SPL {X  -165.650, Y  +571.720, Z    +0.000, E1   +39.004, E3 +431163.246}
SPL {X  -165.650, Y  +565.656, Z    +0.000, E1   +39.042, E3 +431178.355}
SPL {X  -165.650, Y  +560.333, Z    +0.000, E1   +38.995, E3 +431191.984}
SPL {X  -165.650, Y  +554.558, Z    +0.000, E1   +39.065, E3 +431206.273}
SPL {X  -165.650, Y  +548.147, Z    +0.000, E1   +39.104, E3 +431222.129}
SPL {X  -165.650, Y  +526.098, Z    +0.000, E1   +45.792, E3 +431231.948}
SPL {X  -165.650, Y  +510.223, Z    +0.000, E1   +49.521, E3 +431239.345}
SPL {X  -165.650, Y  +506.429, Z    +0.000, E1   +48.913, E3 +431249.758}
SPL {X  -165.650, Y  +501.394, Z    +0.000, E1   +48.110, E3 +431263.737}
SPL {X  -165.650, Y  +497.138, Z    +0.000, E1   +47.280, E3 +431276.433}
SPL {X  -165.650, Y  +493.273, Z    +0.000, E1   +46.518, E3 +431288.414}
SPL {X  -165.650, Y  +489.140, Z    +0.000, E1   +45.675, E3 +431301.541}
SPL {X  -165.650, Y  +485.420, Z    +0.000, E1   +44.711, E3 +431314.760}
SPL {X  -165.650, Y  +480.756, Z    +0.000, E1   +43.779, E3 +431330.238}
SPL {X  -165.650, Y  +475.837, Z    +0.000, E1   +42.787, E3 +431346.699}
SPL {X  -165.650, Y  +472.413, Z    +0.000, E1   +41.852, E3 +431359.813}
SPL {X  -165.650, Y  +468.649, Z    +0.000, E1   +41.090, E3 +431373.177}
SPL {X  -165.650, Y  +465.438, Z    +0.000, E1   +39.745, E3 +431388.974}
ENDSPLINE

SPLINE
SPL {X  -165.650, Y  +478.843, Z    +0.000, E1   +30.924, E3 +431405.859}
ENDSPLINE

SPLINE
SPL {X  -165.650, Y  +474.473, Z    +0.000, E1   +30.943, E3 +431420.492}
SPL {X  -165.650, Y  +470.376, Z    +0.000, E1   +30.888, E3 +431435.022}
SPL {X  -165.650, Y  +465.146, Z    +0.000, E1   +30.883, E3 +431452.952}
SPL {X  -165.650, Y  +461.106, Z    +0.000, E1   +30.916, E3 +431466.370}
SPL {X  -165.650, Y  +457.156, Z    +0.000, E1   +30.860, E3 +431480.446}
SPL {X  -165.650, Y  +453.156, Z    +0.000, E1   +30.934, E3 +431493.420}
SPL {X  -165.650, Y  +450.433, Z    +0.000, E1   +30.789, E3 +431503.776}
SPL {X  -165.650, Y  +447.097, Z    +0.000, E1   +30.843, E3 +431514.824}
SPL {X  -165.650, Y  +443.673, Z    +0.000, E1   +30.907, E3 +431526.132}
SPL {X  -165.650, Y  +439.486, Z    +0.000, E1   +30.857, E3 +431540.941}
SPL {X  -165.650, Y  +435.146, Z    +0.000, E1   +30.969, E3 +431554.861}
SPL {X  -165.650, Y  +432.765, Z    +0.000, E1   +30.831, E3 +431563.875}
SPL {X  -165.650, Y  +429.309, Z    +0.000, E1   +30.920, E3 +431575.216}
SPL {X  -165.650, Y  +424.918, Z    +0.000, E1   +30.862, E3 +431590.673}
SPL {X  -165.650, Y  +421.437, Z    +0.000, E1   +30.833, E3 +431602.641}
SPL {X  -165.650, Y  +417.366, Z    +0.000, E1   +30.879, E3 +431616.482}
SPL {X  -165.650, Y  +413.181, Z    +0.000, E1   +30.815, E3 +431631.079}
SPL {X  -165.650, Y  +408.547, Z    +0.000, E1   +30.964, E3 +431646.082}
SPL {X  -165.650, Y  +403.421, Z    +0.000, E1   +30.863, E3 +431664.300}
SPL {X  -165.650, Y  +398.147, Z    +0.000, E1   +30.902, E3 +431682.061}
SPL {X  -165.650, Y  +394.694, Z    +0.000, E1   +30.805, E3 +431694.369}
SPL {X  -165.650, Y  +390.331, Z    +0.000, E1   +30.892, E3 +431708.945}
SPL {X  -165.650, Y  +384.849, Z    +0.000, E1   +30.885, E3 +431727.748}
SPL {X  -165.650, Y  +380.752, Z    +0.000, E1   +30.927, E3 +431741.250}
SPL {X  -165.648, Y  +377.739, Z    +0.000, E1   +30.835, E3 +431752.260}
SPL {X  -165.594, Y  +374.183, Z    +0.000, E1   +30.878, E3 +431764.096}
SPL {X  -165.429, Y  +369.945, Z    +0.000, E1   +30.850, E3 +431778.972}
SPL {X  -165.167, Y  +365.866, Z    +0.000, E1   +30.741, E3 +431793.504}
SPL {X  -164.892, Y  +362.671, Z    +0.000, E1   +30.830, E3 +431803.828}
SPL {X  -164.570, Y  +359.612, Z    +0.000, E1   +30.773, E3 +431814.641}
SPL {X  -164.287, Y  +357.291, Z    +0.000, E1   +30.513, E3 +431824.270}
SPL {X  -163.720, Y  +353.284, Z    +0.000, E1   +30.592, E3 +431837.717}
SPL {X  -162.976, Y  +348.856, Z    +0.000, E1   +30.757, E3 +431851.546}
SPL {X  -161.497, Y  +341.640, Z    +0.000, E1   +33.276, E3 +431858.823}
SPL {X  -152.976, Y  +314.952, Z    +0.000, E1   +38.607, E3 +431903.168}
SPL {X  -137.967, Y  +286.821, Z    +0.000, E1   +43.969, E3 +431946.389}
ENDSPLINE

SPLINE
SPL {X  -149.143, Y  +306.414, Z    +0.000, E1   +36.361, E3 +431997.522}
SPL {X  -163.091, Y  +349.496, Z    +0.000, E1   +19.699, E3 +431954.305}
SPL {X  -165.027, Y  +364.142, Z    +0.000, E1   +12.054, E3 +431957.445}
SPL {X  -165.612, Y  +374.969, Z    +0.000, E1    +5.630, E3 +431962.628}
SPL {X  -165.650, Y  +383.362, Z    +0.000, E1    +0.177, E3 +431947.246}
SPL {X  -165.650, Y  +383.923, Z    +0.000, E1    -0.215, E3 +431960.404}
SPL {X  -165.650, Y  +388.083, Z    +0.000, E1    -3.355, E3 +431959.267}
SPL {X  -165.650, Y  +395.510, Z    +0.000, E1    -9.810, E3 +431955.393}
SPL {X  -165.650, Y  +403.066, Z    +0.000, E1   -17.886, E3 +431948.226}
SPL {X  -165.650, Y  +414.811, Z    +0.000, E1   -28.314, E3 +431949.707}
SPL {X  -165.650, Y  +423.479, Z    +0.000, E1   -29.012, E3 +431973.636}
SPL {X  -165.650, Y  +441.276, Z    +0.000, E1   -37.343, E3 +431985.325}
SPL {X  -165.650, Y  +462.890, Z    +0.000, E1   -40.484, E3 +432019.408}
ENDSPLINE

SPLINE
SPL {X  -165.650, Y  +446.920, Z    +0.000, E1   -31.238, E3 +432031.734}
ENDSPLINE

SPLINE
SPL {X  -165.650, Y  +447.935, Z    +0.000, E1   -30.213, E3 +432042.022}
SPL {X  -165.650, Y  +451.020, Z    +0.000, E1   -30.224, E3 +432052.842}
SPL {X  -165.650, Y  +454.519, Z    +0.000, E1   -30.374, E3 +432064.024}
SPL {X  -165.650, Y  +456.542, Z    +0.000, E1   -29.986, E3 +432073.769}
SPL {X  -165.650, Y  +460.618, Z    +0.000, E1   -30.298, E3 +432086.090}
SPL {X  -165.650, Y  +463.853, Z    +0.000, E1   -30.103, E3 +432098.690}
SPL {X  -165.650, Y  +468.397, Z    +0.000, E1   -30.302, E3 +432113.494}
SPL {X  -165.650, Y  +472.566, Z    +0.000, E1   -30.124, E3 +432129.204}
SPL {X  -165.650, Y  +475.265, Z    +0.000, E1   -30.034, E3 +432139.241}
SPL {X  -165.650, Y  +479.559, Z    +0.000, E1   -30.258, E3 +432153.106}
SPL {X  -165.650, Y  +484.477, Z    +0.000, E1   -30.274, E3 +432170.115}
SPL {X  -165.650, Y  +488.041, Z    +0.000, E1   -30.253, E3 +432182.670}
SPL {X  -165.650, Y  +491.281, Z    +0.000, E1   -30.148, E3 +432194.808}
SPL {X  -165.650, Y  +495.051, Z    +0.000, E1   -30.213, E3 +432207.617}
SPL {X  -165.650, Y  +499.546, Z    +0.000, E1   -30.283, E3 +432223.059}
SPL {X  -165.650, Y  +503.544, Z    +0.000, E1   -30.247, E3 +432237.128}
SPL {X  -165.650, Y  +506.344, Z    +0.000, E1   -30.129, E3 +432247.797}
SPL {X  -165.650, Y  +509.866, Z    +0.000, E1   -30.236, E3 +432259.466}
SPL {X  -165.650, Y  +513.685, Z    +0.000, E1   -30.234, E3 +432272.962}
SPL {X  -165.650, Y  +517.919, Z    +0.000, E1   -30.227, E3 +432287.869}
SPL {X  -165.650, Y  +521.521, Z    +0.000, E1   -30.210, E3 +432300.544}
SPL {X  -165.650, Y  +525.344, Z    +0.000, E1   -30.269, E3 +432313.650}
SPL {X  -165.650, Y  +528.152, Z    +0.000, E1   -29.991, E3 +432325.291}
SPL {X  -165.650, Y  +531.783, Z    +0.000, E1   -30.416, E3 +432335.184}
SPL {X  -165.650, Y  +534.115, Z    +0.000, E1   -30.089, E3 +432345.566}
SPL {X  -165.650, Y  +537.522, Z    +0.000, E1   -30.251, E3 +432356.480}
SPL {X  -165.650, Y  +540.621, Z    +0.000, E1   -30.014, E3 +432369.041}
SPL {X  -165.650, Y  +544.944, Z    +0.000, E1   -30.447, E3 +432381.241}
SPL {X  -165.650, Y  +547.199, Z    +0.000, E1   -30.132, E3 +432391.214}
SPL {X  -165.650, Y  +550.512, Z    +0.000, E1   -30.197, E3 +432402.540}
SPL {X  -165.650, Y  +553.852, Z    +0.000, E1   -30.156, E3 +432414.481}
SPL {X  -165.650, Y  +557.277, Z    +0.000, E1   -30.150, E3 +432426.655}
SPL {X  -165.650, Y  +561.168, Z    +0.000, E1   -30.194, E3 +432440.037}
SPL {X  -165.650, Y  +565.528, Z    +0.000, E1   -30.192, E3 +432455.520}
SPL {X  -165.650, Y  +570.048, Z    +0.000, E1   -30.238, E3 +432470.951}
SPL {X  -165.650, Y  +573.110, Z    +0.000, E1   -30.057, E3 +432482.936}
SPL {X  -165.650, Y  +577.587, Z    +0.000, E1   -30.270, E3 +432497.375}
SPL {X  -165.650, Y  +581.190, Z    +0.000, E1   -30.107, E3 +432511.014}
SPL {X  -165.650, Y  +585.053, Z    +0.000, E1   -30.090, E3 +432524.884}
ENDSPLINE

SPLINE
SPL {X  -165.650, Y  +484.445, Z    +0.000, E1   +32.277, E3 +432542.289}
SPL {X  -165.650, Y  +481.524, Z    +0.000, E1   +31.089, E3 +432559.739}
SPL {X  -165.650, Y  +478.014, Z    +0.000, E1   +30.826, E3 +432573.347}
SPL {X  -165.650, Y  +474.473, Z    +0.000, E1   +30.943, E3 +432584.671}
SPL {X  -165.650, Y  +471.826, Z    +0.000, E1   +30.770, E3 +432594.855}
SPL {X  -165.650, Y  +467.753, Z    +0.000, E1   +30.878, E3 +432608.228}
SPL {X  -165.650, Y  +463.837, Z    +0.000, E1   +30.924, E3 +432621.162}
SPL {X  -165.650, Y  +461.106, Z    +0.000, E1   +30.916, E3 +432630.549}
SPL {X  -165.650, Y  +457.156, Z    +0.000, E1   +30.860, E3 +432644.626}
SPL {X  -165.650, Y  +453.156, Z    +0.000, E1   +30.934, E3 +432657.600}
SPL {X  -165.650, Y  +450.433, Z    +0.000, E1   +30.789, E3 +432667.955}
SPL {X  -165.650, Y  +447.097, Z    +0.000, E1   +30.843, E3 +432679.004}
SPL {X  -165.650, Y  +443.673, Z    +0.000, E1   +30.907, E3 +432690.311}
SPL {X  -165.650, Y  +439.486, Z    +0.000, E1   +30.857, E3 +432705.120}
SPL {X  -165.650, Y  +435.146, Z    +0.000, E1   +30.969, E3 +432719.040}
SPL {X  -165.650, Y  +432.765, Z    +0.000, E1   +30.831, E3 +432728.054}
SPL {X  -165.650, Y  +429.309, Z    +0.000, E1   +30.920, E3 +432739.395}
SPL {X  -165.650, Y  +424.918, Z    +0.000, E1   +30.862, E3 +432754.852}
SPL {X  -165.650, Y  +421.437, Z    +0.000, E1   +30.833, E3 +432766.820}
SPL {X  -165.650, Y  +417.366, Z    +0.000, E1   +30.879, E3 +432780.661}
SPL {X  -165.650, Y  +413.181, Z    +0.000, E1   +30.815, E3 +432795.259}
SPL {X  -165.650, Y  +408.547, Z    +0.000, E1   +30.964, E3 +432810.261}
SPL {X  -165.650, Y  +405.433, Z    +0.000, E1   +30.730, E3 +432822.239}
SPL {X  -165.650, Y  +402.516, Z    +0.000, E1   +30.874, E3 +432831.361}
SPL {X  -165.650, Y  +398.147, Z    +0.000, E1   +30.902, E3 +432846.240}
SPL {X  -165.650, Y  +394.694, Z    +0.000, E1   +30.805, E3 +432858.548}
SPL {X  -165.650, Y  +391.522, Z    +0.000, E1   +30.837, E3 +432869.229}
SPL {X  -165.650, Y  +387.533, Z    +0.000, E1   +30.858, E3 +432882.855}
SPL {X  -165.650, Y  +383.627, Z    +0.000, E1   +30.885, E3 +432895.915}
SPL {X  -165.650, Y  +380.752, Z    +0.000, E1   +30.927, E3 +432905.429}
SPL {X  -165.648, Y  +377.739, Z    +0.000, E1   +30.835, E3 +432916.439}
SPL {X  -165.594, Y  +374.183, Z    +0.000, E1   +30.878, E3 +432928.276}
SPL {X  -165.429, Y  +369.945, Z    +0.000, E1   +30.850, E3 +432943.151}
SPL {X  -165.167, Y  +365.866, Z    +0.000, E1   +30.741, E3 +432957.683}
SPL {X  -164.892, Y  +362.671, Z    +0.000, E1   +30.830, E3 +432968.007}
SPL {X  -164.570, Y  +359.612, Z    +0.000, E1   +30.773, E3 +432978.820}
SPL {X  -164.104, Y  +355.923, Z    +0.000, E1   +30.626, E3 +432992.536}
SPL {X  -163.573, Y  +352.353, Z    +0.000, E1   +30.451, E3 +433005.801}
SPL {X  -162.476, Y  +346.230, Z    +0.000, E1   +31.677, E3 +433018.382}
SPL {X  -152.976, Y  +314.952, Z    +0.000, E1   +38.607, E3 +433067.347}
SPL {X  -137.967, Y  +286.821, Z    +0.000, E1   +43.969, E3 +433110.568}
ENDSPLINE

SPLINE
SPL {X  -149.143, Y  +306.414, Z    +0.000, E1   +36.361, E3 +433161.701}
SPL {X  -164.268, Y  +357.145, Z    +0.000, E1   +15.880, E3 +433119.460}
SPL {X  -165.379, Y  +369.025, Z    +0.000, E1    +9.158, E3 +433124.131}
SPL {X  -165.612, Y  +374.969, Z    +0.000, E1    +5.630, E3 +433126.807}
SPL {X  -165.650, Y  +383.362, Z    +0.000, E1    +0.177, E3 +433111.425}
SPL {X  -165.650, Y  +383.923, Z    +0.000, E1    -0.215, E3 +433124.583}
SPL {X  -165.650, Y  +388.083, Z    +0.000, E1    -3.355, E3 +433123.446}
SPL {X  -165.650, Y  +393.983, Z    +0.000, E1    -8.501, E3 +433119.844}
SPL {X  -165.650, Y  +402.241, Z    +0.000, E1   -16.711, E3 +433114.356}
SPL {X  -165.650, Y  +416.345, Z    +0.000, E1   -29.511, E3 +433114.148}
SPL {X  -165.650, Y  +422.331, Z    +0.000, E1   -27.760, E3 +433139.647}
SPL {X  -165.650, Y  +441.276, Z    +0.000, E1   -37.343, E3 +433149.504}
SPL {X  -165.650, Y  +462.890, Z    +0.000, E1   -40.484, E3 +433183.587}
ENDSPLINE

SPLINE
SPL {X  -165.650, Y  +446.920, Z    +0.000, E1   -31.238, E3 +433195.913}
ENDSPLINE

SPLINE
SPL {X  -165.650, Y  +447.935, Z    +0.000, E1   -30.213, E3 +433206.201}
SPL {X  -165.650, Y  +451.020, Z    +0.000, E1   -30.224, E3 +433217.021}
SPL {X  -165.650, Y  +454.519, Z    +0.000, E1   -30.374, E3 +433228.204}
SPL {X  -165.650, Y  +457.429, Z    +0.000, E1   -30.029, E3 +433240.905}
SPL {X  -165.650, Y  +461.678, Z    +0.000, E1   -30.426, E3 +433253.030}
SPL {X  -165.650, Y  +463.853, Z    +0.000, E1   -30.103, E3 +433262.870}
SPL {X  -165.650, Y  +468.397, Z    +0.000, E1   -30.302, E3 +433277.673}
SPL {X  -165.650, Y  +472.566, Z    +0.000, E1   -30.124, E3 +433293.383}
SPL {X  -165.650, Y  +475.265, Z    +0.000, E1   -30.034, E3 +433303.420}
SPL {X  -165.650, Y  +477.862, Z    +0.000, E1   -30.319, E3 +433310.612}
SPL {X  -165.650, Y  +481.042, Z    +0.000, E1   -30.192, E3 +433322.872}
SPL {X  -165.650, Y  +485.236, Z    +0.000, E1   -30.294, E3 +433336.728}
SPL {X  -165.650, Y  +488.041, Z    +0.000, E1   -30.253, E3 +433346.849}
SPL {X  -165.650, Y  +491.281, Z    +0.000, E1   -30.148, E3 +433358.987}
SPL {X  -165.650, Y  +495.051, Z    +0.000, E1   -30.213, E3 +433371.796}
SPL {X  -165.650, Y  +499.546, Z    +0.000, E1   -30.283, E3 +433387.239}
SPL {X  -165.650, Y  +503.544, Z    +0.000, E1   -30.247, E3 +433401.307}
SPL {X  -165.650, Y  +506.344, Z    +0.000, E1   -30.129, E3 +433411.976}
SPL {X  -165.650, Y  +509.866, Z    +0.000, E1   -30.236, E3 +433423.645}
SPL {X  -165.650, Y  +513.685, Z    +0.000, E1   -30.234, E3 +433437.141}
SPL {X  -165.650, Y  +517.919, Z    +0.000, E1   -30.227, E3 +433452.048}
SPL {X  -165.650, Y  +521.521, Z    +0.000, E1   -30.210, E3 +433464.723}
SPL {X  -165.650, Y  +525.344, Z    +0.000, E1   -30.269, E3 +433477.829}
SPL {X  -165.650, Y  +528.152, Z    +0.000, E1   -29.991, E3 +433489.470}
SPL {X  -165.650, Y  +531.783, Z    +0.000, E1   -30.416, E3 +433499.363}
SPL {X  -165.650, Y  +534.115, Z    +0.000, E1   -30.089, E3 +433509.745}
SPL {X  -165.650, Y  +537.522, Z    +0.000, E1   -30.251, E3 +433520.659}
SPL {X  -165.650, Y  +540.621, Z    +0.000, E1   -30.014, E3 +433533.220}
SPL {X  -165.650, Y  +544.944, Z    +0.000, E1   -30.447, E3 +433545.420}
SPL {X  -165.650, Y  +547.199, Z    +0.000, E1   -30.132, E3 +433555.394}
SPL {X  -165.650, Y  +550.512, Z    +0.000, E1   -30.197, E3 +433566.719}
SPL {X  -165.650, Y  +553.852, Z    +0.000, E1   -30.156, E3 +433578.660}
SPL {X  -165.650, Y  +557.277, Z    +0.000, E1   -30.150, E3 +433590.835}
SPL {X  -165.650, Y  +561.168, Z    +0.000, E1   -30.194, E3 +433604.216}
SPL {X  -165.650, Y  +564.449, Z    +0.000, E1   -30.167, E3 +433615.899}
SPL {X  -165.650, Y  +566.935, Z    +0.000, E1   -30.135, E3 +433624.805}
SPL {X  -165.650, Y  +570.048, Z    +0.000, E1   -30.238, E3 +433635.130}
SPL {X  -165.650, Y  +573.110, Z    +0.000, E1   -30.057, E3 +433647.115}
SPL {X  -165.650, Y  +577.587, Z    +0.000, E1   -30.270, E3 +433661.554}
SPL {X  -165.650, Y  +581.190, Z    +0.000, E1   -30.107, E3 +433675.193}
SPL {X  -165.650, Y  +585.053, Z    +0.000, E1   -30.090, E3 +433689.063}
ENDSPLINE

SPLINE
SPL {X  -165.650, Y  +484.445, Z    +0.000, E1   +32.277, E3 +433706.468}
SPL {X  -165.650, Y  +481.524, Z    +0.000, E1   +31.089, E3 +433723.918}
SPL {X  -165.650, Y  +478.014, Z    +0.000, E1   +30.826, E3 +433737.526}
SPL {X  -165.650, Y  +474.473, Z    +0.000, E1   +30.943, E3 +433748.850}
SPL {X  -165.650, Y  +471.826, Z    +0.000, E1   +30.770, E3 +433759.034}
SPL {X  -165.650, Y  +467.753, Z    +0.000, E1   +30.878, E3 +433772.407}
SPL {X  -165.650, Y  +463.837, Z    +0.000, E1   +30.924, E3 +433785.341}
SPL {X  -165.650, Y  +461.106, Z    +0.000, E1   +30.916, E3 +433794.728}
SPL {X  -165.650, Y  +457.156, Z    +0.000, E1   +30.860, E3 +433808.805}
SPL {X  -165.650, Y  +453.156, Z    +0.000, E1   +30.934, E3 +433821.779}
SPL {X  -165.650, Y  +450.433, Z    +0.000, E1   +30.789, E3 +433832.134}
SPL {X  -165.650, Y  +447.097, Z    +0.000, E1   +30.843, E3 +433843.183}
SPL {X  -165.650, Y  +443.673, Z    +0.000, E1   +30.907, E3 +433854.490}
SPL {X  -165.650, Y  +439.486, Z    +0.000, E1   +30.857, E3 +433869.299}
SPL {X  -165.650, Y  +435.146, Z    +0.000, E1   +30.969, E3 +433883.219}
SPL {X  -165.650, Y  +431.607, Z    +0.000, E1   +30.889, E3 +433895.933}
SPL {X  -165.650, Y  +427.340, Z    +0.000, E1   +30.870, E3 +433910.645}
SPL {X  -165.650, Y  +423.901, Z    +0.000, E1   +30.858, E3 +433922.401}
SPL {X  -165.650, Y  +421.437, Z    +0.000, E1   +30.833, E3 +433931.000}
SPL {X  -165.650, Y  +418.489, Z    +0.000, E1   +30.835, E3 +433941.116}
SPL {X  -165.650, Y  +414.127, Z    +0.000, E1   +30.869, E3 +433956.025}
SPL {X  -165.650, Y  +408.547, Z    +0.000, E1   +30.964, E3 +433974.440}
SPL {X  -165.650, Y  +405.433, Z    +0.000, E1   +30.730, E3 +433986.418}
SPL {X  -165.650, Y  +401.473, Z    +0.000, E1   +30.933, E3 +433998.866}
SPL {X  -165.650, Y  +396.018, Z    +0.000, E1   +30.861, E3 +434018.051}
SPL {X  -165.650, Y  +391.522, Z    +0.000, E1   +30.837, E3 +434033.408}
SPL {X  -165.650, Y  +387.533, Z    +0.000, E1   +30.858, E3 +434047.034}
SPL {X  -165.650, Y  +383.627, Z    +0.000, E1   +30.885, E3 +434060.094}
SPL {X  -165.650, Y  +380.752, Z    +0.000, E1   +30.927, E3 +434069.608}
SPL {X  -165.648, Y  +377.739, Z    +0.000, E1   +30.835, E3 +434080.618}
SPL {X  -165.594, Y  +374.183, Z    +0.000, E1   +30.878, E3 +434092.455}
SPL {X  -165.429, Y  +369.945, Z    +0.000, E1   +30.850, E3 +434107.330}
SPL {X  -165.167, Y  +365.866, Z    +0.000, E1   +30.741, E3 +434121.862}
SPL {X  -164.892, Y  +362.671, Z    +0.000, E1   +30.830, E3 +434132.186}
SPL {X  -164.570, Y  +359.612, Z    +0.000, E1   +30.773, E3 +434142.999}
SPL {X  -164.104, Y  +355.923, Z    +0.000, E1   +30.626, E3 +434156.716}
SPL {X  -163.573, Y  +352.353, Z    +0.000, E1   +30.451, E3 +434169.980}
SPL {X  -162.976, Y  +348.856, Z    +0.000, E1   +30.757, E3 +434179.904}
SPL {X  -161.497, Y  +341.640, Z    +0.000, E1   +33.276, E3 +434187.182}
SPL {X  -152.976, Y  +314.952, Z    +0.000, E1   +38.607, E3 +434231.526}
SPL {X  -137.967, Y  +286.821, Z    +0.000, E1   +43.969, E3 +434274.747}
ENDSPLINE

SPLINE
SPL {X  -149.143, Y  +306.414, Z    +0.000, E1   +36.361, E3 +434325.880}
SPL {X  -164.268, Y  +357.145, Z    +0.000, E1   +15.880, E3 +434283.639}
SPL {X  -165.510, Y  +371.680, Z    +0.000, E1    +7.684, E3 +434286.641}
SPL {X  -165.628, Y  +375.818, Z    +0.000, E1    +5.016, E3 +434294.571}
SPL {X  -165.650, Y  +383.362, Z    +0.000, E1    +0.177, E3 +434275.604}
SPL {X  -165.650, Y  +383.923, Z    +0.000, E1    -0.215, E3 +434288.762}
SPL {X  -165.650, Y  +388.083, Z    +0.000, E1    -3.355, E3 +434287.625}
SPL {X  -165.650, Y  +395.510, Z    +0.000, E1    -9.810, E3 +434283.751}
SPL {X  -165.650, Y  +403.066, Z    +0.000, E1   -17.886, E3 +434276.584}
SPL {X  -165.650, Y  +416.345, Z    +0.000, E1   -29.511, E3 +434278.327}
SPL {X  -165.650, Y  +422.331, Z    +0.000, E1   -27.760, E3 +434303.826}
SPL {X  -165.650, Y  +441.276, Z    +0.000, E1   -37.343, E3 +434313.683}
SPL {X  -165.650, Y  +462.890, Z    +0.000, E1   -40.484, E3 +434347.766}
ENDSPLINE

SPLINE
SPL {X  -165.650, Y  +446.920, Z    +0.000, E1   -31.238, E3 +434360.092}
ENDSPLINE

SPLINE
SPL {X  -165.650, Y  +447.935, Z    +0.000, E1   -30.213, E3 +434370.380}
SPL {X  -165.650, Y  +451.020, Z    +0.000, E1   -30.224, E3 +434381.200}
SPL {X  -165.650, Y  +454.519, Z    +0.000, E1   -30.374, E3 +434392.383}
SPL {X  -165.650, Y  +457.429, Z    +0.000, E1   -30.029, E3 +434405.084}
SPL {X  -165.650, Y  +461.678, Z    +0.000, E1   -30.426, E3 +434417.209}
SPL {X  -165.650, Y  +463.853, Z    +0.000, E1   -30.103, E3 +434427.049}
SPL {X  -165.650, Y  +468.397, Z    +0.000, E1   -30.302, E3 +434441.853}
SPL {X  -165.650, Y  +472.566, Z    +0.000, E1   -30.124, E3 +434457.562}
SPL {X  -165.650, Y  +475.265, Z    +0.000, E1   -30.034, E3 +434467.599}
SPL {X  -165.650, Y  +477.862, Z    +0.000, E1   -30.319, E3 +434474.791}
SPL {X  -165.650, Y  +481.042, Z    +0.000, E1   -30.192, E3 +434487.051}
SPL {X  -165.650, Y  +485.236, Z    +0.000, E1   -30.294, E3 +434500.907}
SPL {X  -165.650, Y  +488.041, Z    +0.000, E1   -30.253, E3 +434511.028}
SPL {X  -165.650, Y  +491.281, Z    +0.000, E1   -30.148, E3 +434523.166}
SPL {X  -165.650, Y  +495.051, Z    +0.000, E1   -30.213, E3 +434535.975}
SPL {X  -165.650, Y  +499.546, Z    +0.000, E1   -30.283, E3 +434551.418}
SPL {X  -165.650, Y  +503.544, Z    +0.000, E1   -30.247, E3 +434565.486}
SPL {X  -165.650, Y  +506.344, Z    +0.000, E1   -30.129, E3 +434576.155}
SPL {X  -165.650, Y  +510.660, Z    +0.000, E1   -30.223, E3 +434590.858}
SPL {X  -165.650, Y  +514.670, Z    +0.000, E1   -30.278, E3 +434604.368}
SPL {X  -165.650, Y  +517.919, Z    +0.000, E1   -30.227, E3 +434616.227}
SPL {X  -165.650, Y  +522.822, Z    +0.000, E1   -30.289, E3 +434633.117}
SPL {X  -165.650, Y  +527.393, Z    +0.000, E1   -30.104, E3 +434650.365}
SPL {X  -165.650, Y  +531.783, Z    +0.000, E1   -30.416, E3 +434663.542}
SPL {X  -165.650, Y  +534.115, Z    +0.000, E1   -30.089, E3 +434673.924}
SPL {X  -165.650, Y  +537.522, Z    +0.000, E1   -30.251, E3 +434684.838}
SPL {X  -165.650, Y  +540.621, Z    +0.000, E1   -30.014, E3 +434697.399}
SPL {X  -165.650, Y  +544.944, Z    +0.000, E1   -30.447, E3 +434709.599}
SPL {X  -165.650, Y  +547.199, Z    +0.000, E1   -30.132, E3 +434719.573}
SPL {X  -165.650, Y  +550.512, Z    +0.000, E1   -30.197, E3 +434730.898}
SPL {X  -165.650, Y  +553.852, Z    +0.000, E1   -30.156, E3 +434742.839}
SPL {X  -165.650, Y  +557.277, Z    +0.000, E1   -30.150, E3 +434755.014}
SPL {X  -165.650, Y  +561.168, Z    +0.000, E1   -30.194, E3 +434768.395}
SPL {X  -165.650, Y  +565.528, Z    +0.000, E1   -30.192, E3 +434783.878}
SPL {X  -165.650, Y  +570.048, Z    +0.000, E1   -30.238, E3 +434799.309}
SPL {X  -165.650, Y  +573.110, Z    +0.000, E1   -30.057, E3 +434811.294}
SPL {X  -165.650, Y  +577.587, Z    +0.000, E1   -30.270, E3 +434825.733}
SPL {X  -165.650, Y  +581.190, Z    +0.000, E1   -30.107, E3 +434839.372}
SPL {X  -165.650, Y  +585.053, Z    +0.000, E1   -30.090, E3 +434853.242}
ENDSPLINE

